cylinder.List.fbAllocateRobot_LeftClamp1(xDone =>,
                                         xBusy =>,
                                         xError =>CylinderStatus.AllocateRobot_LeftClamp1.Error,
                                         xEnable :=,
                                         FrontSensor :=,
                                         RearSensor :=,
                                         SetupPara := CurrentData.Cylinders.AllocateRobot_LeftClamp1,
                                         CurrentCylinderType =>,
                                         InFrontPosition =>CylinderStatus.AllocateRobot_LeftClamp1.InFrontPosition,
                                         InRearPosition =>CylinderStatus.AllocateRobot_LeftClamp1.InRearPosition,
                                         ExtendOutput => InternalOutput.bAllocateRobot_LeftClamp1_Close_Valve,
                                         RetractOutput => InternalOutput.bAllocateRobot_LeftClamp1_Open_Valve);
cylinder.List.fbAllocateRobot_LeftClamp1.IsDoubleValve := TRUE;

cylinder.List.fbAllocateRobot_LeftClamp2(xDone =>,
                                         xBusy =>,
                                         xError =>CylinderStatus.AllocateRobot_LeftClamp2.Error,
                                         xEnable :=,
                                         FrontSensor :=,
                                         RearSensor :=,
                                         SetupPara := CurrentData.Cylinders.AllocateRobot_LeftClamp2,
                                         CurrentCylinderType =>,
                                         InFrontPosition =>CylinderStatus.AllocateRobot_LeftClamp2.InFrontPosition,
                                         InRearPosition =>CylinderStatus.AllocateRobot_LeftClamp2.InRearPosition,
                                         ExtendOutput => InternalOutput.bAllocateRobot_LeftClamp2_Close_Valve,
                                         RetractOutput => InternalOutput.bAllocateRobot_LeftClamp2_Open_Valve);
cylinder.List.fbAllocateRobot_LeftClamp2.IsDoubleValve := TRUE;

cylinder.List.fbAllocateRobot_RightClamp1(xDone =>,
                                          xBusy =>,
                                          xError =>CylinderStatus.AllocateRobot_RightClamp1.Error,
                                          xEnable :=,
                                          FrontSensor :=,
                                          RearSensor :=,
                                          SetupPara := CurrentData.Cylinders.AllocateRobot_RightClamp1,
                                          CurrentCylinderType =>,
                                          InFrontPosition =>CylinderStatus.AllocateRobot_RightClamp1.InFrontPosition,
                                          InRearPosition =>CylinderStatus.AllocateRobot_RightClamp1.InRearPosition,
                                          ExtendOutput => InternalOutput.bAllocateRobot_RightClamp1_Close_Valve,
                                          RetractOutput => InternalOutput.bAllocateRobot_RightClamp1_Open_Valve);
cylinder.List.fbAllocateRobot_RightClamp1.IsDoubleValve := TRUE;

cylinder.List.fbAllocateRobot_RightClamp2(xDone =>,
                                          xBusy =>,
                                          xError =>CylinderStatus.AllocateRobot_RightClamp2.Error,
                                          xEnable :=,
                                          FrontSensor :=,
                                          RearSensor :=,
                                          SetupPara := CurrentData.Cylinders.AllocateRobot_RightClamp2,
                                          CurrentCylinderType =>,
                                          InFrontPosition =>CylinderStatus.AllocateRobot_RightClamp2.InFrontPosition,
                                          InRearPosition =>CylinderStatus.AllocateRobot_RightClamp2.InRearPosition,
                                          ExtendOutput => InternalOutput.bAllocateRobot_RightClamp2_Close_Valve,
                                          RetractOutput => InternalOutput.bAllocateRobot_RightClamp2_Open_Valve);
cylinder.List.fbAllocateRobot_RightClamp2.IsDoubleValve := TRUE;

cylinder.List.fbRoundBelt_WorkZone_Press(xDone =>,
                                         xBusy =>,
                                         xError =>CylinderStatus.RoundBelt_WorkZone_Press.Error,
                                         xEnable :=,
                                         FrontSensor :=,
                                         RearSensor := input.bRoundBelt_WorkZonePress_RearSensor,
                                         SetupPara := CurrentData.Cylinders.RoundBelt_WorkZone_Press,
                                         CurrentCylinderType =>,
                                         InFrontPosition =>CylinderStatus.RoundBelt_WorkZone_Press.InFrontPosition,
                                         InRearPosition =>CylinderStatus.RoundBelt_WorkZone_Press.InRearPosition,
                                         ExtendOutput => InternalOutput.bRoundBelt_WorkZone_Press_Valve,
                                         RetractOutput =>);

cylinder.List.fbRoundBelt_WorkZone_Plug(xDone =>,
                                        xBusy =>,
                                        xError =>CylinderStatus.RoundBelt_WorkZone_Plug.Error,
                                        xEnable :=,
                                        FrontSensor := input.bRoundBelt_WorkZonePlug_frontSensor,
                                        RearSensor := INPUT.bRoundBelt_WorkZonePlug_RearSensor,
                                        SetupPara := CurrentData.Cylinders.RoundBelt_WorkZone_Plug,
                                        CurrentCylinderType =>,
                                        InFrontPosition =>CylinderStatus.RoundBelt_WorkZone_Plug.InFrontPosition,
                                        InRearPosition =>CylinderStatus.RoundBelt_WorkZone_Plug.InRearPosition,
                                        ExtendOutput => InternalOutput.bRoundBelt_WorkZone_Plug_Valve,
                                        RetractOutput =>);

cylinder.List.fbRoundBelt_ChargeZone_Plug(xDone =>,
                                          xBusy =>,
                                          xError =>CylinderStatus.RoundBelt_ChargeZone_Plug.Error,
                                          xEnable :=,
                                          FrontSensor := INPUT.bRoundBelt_ChangeZonePlug_FrontSensor,
                                          RearSensor := input.bRoundBelt_ChangeZonePlug_RearSensor,
                                          SetupPara := CurrentData.Cylinders.RoundBelt_ChargeZone_Plug,
                                          CurrentCylinderType =>,
                                          InFrontPosition =>CylinderStatus.RoundBelt_ChargeZone_Plug.InFrontPosition,
                                          InRearPosition =>CylinderStatus.RoundBelt_ChargeZone_Plug.InRearPosition,
                                          ExtendOutput => InternalOutput.bRoundBelt_ChargeZone_Plug_Valve,
                                          RetractOutput =>);

cylinder.List.fbRoundBelt_TransmitCVZone_Plug(xDone =>,
                                              xBusy =>,
                                              xError =>CylinderStatus.RoundBelt_TransmitCVZone_Plug.Error,
                                              xEnable :=,
                                              FrontSensor := input.bRoundBelt_TransmitCVZonePlug_FrontSensor,
                                              RearSensor := INPUT.bRoundBelt_TransmitCVZonePlug_RearSensor,
                                              SetupPara := CurrentData.Cylinders.RoundBelt_TransmitCVZone_Plug,
                                              CurrentCylinderType =>,
                                              InFrontPosition =>CylinderStatus.RoundBelt_TransmitCVZone_Plug.InFrontPosition,
                                              InRearPosition =>CylinderStatus.RoundBelt_TransmitCVZone_Plug.InRearPosition,
                                              ExtendOutput => InternalOutput.bRoundBelt_TransmitCVZone_Plug_Valve,
                                              RetractOutput =>);

cylinder.List.fbOutRobot_AsideVert(xDone =>,
                                   xBusy =>,
                                   xError =>CylinderStatus.OutRobot_AsideVert.Error,
                                   xEnable :=,
                                   FrontSensor := INPUT.bOutRobot_AsideVert_LowSensor,
                                   RearSensor := input.bOutRobot_AsideVert_highSensor,
                                   SetupPara := CurrentData.Cylinders.OutRobot_AsideVert,
                                   CurrentCylinderType =>,
                                   InFrontPosition =>CylinderStatus.OutRobot_AsideVert.InFrontPosition,
                                   InRearPosition =>CylinderStatus.OutRobot_AsideVert.InRearPosition,
                                   ExtendOutput => InternalOutput.bOutRobot_AsideVert_Valve,
                                   RetractOutput =>);

cylinder.List.fbOutRobot_BsideVert(xDone =>,
                                   xBusy =>,
                                   xError =>CylinderStatus.OutRobot_BsideVert.Error,
                                   xEnable :=,
                                   FrontSensor := input.bOutRobot_BsideVert_LowSensor,
                                   RearSensor := INPUT.bOutRobot_BsideVert_HighSensor,
                                   SetupPara := CurrentData.Cylinders.OutRobot_BsideVert,
                                   CurrentCylinderType =>,
                                   InFrontPosition =>CylinderStatus.OutRobot_BsideVert.InFrontPosition,
                                   InRearPosition =>CylinderStatus.OutRobot_BsideVert.InRearPosition,
                                   ExtendOutput => InternalOutput.bOutRobot_BsideVert_Valve,
                                   RetractOutput =>);

cylinder.List.fbOutRobot_AsideClamp(xDone =>,
                                    xBusy =>,
                                    xError =>CylinderStatus.OutRobot_AsideClamp.Error,
                                    xEnable :=,
                                    FrontSensor :=,
                                    RearSensor := input.bOutRobot_AsideClamp_RearSensor,
                                    SetupPara := CurrentData.Cylinders.OutRobot_AsideClamp,
                                    CurrentCylinderType =>,
                                    InFrontPosition =>CylinderStatus.OutRobot_AsideClamp.InFrontPosition,
                                    InRearPosition =>CylinderStatus.OutRobot_AsideClamp.InRearPosition,
                                    ExtendOutput => InternalOutput.bOutRobot_AsideClamp_Close_Valve,
                                    RetractOutput => InternalOutput.bOutRobot_AsideClamp_Open_Valve);
cylinder.List.fbOutRobot_AsideClamp.IsDoubleValve := TRUE;

cylinder.List.fbOutRobot_BsideClamp(xDone =>,
                                    xBusy =>,
                                    xError =>CylinderStatus.OutRobot_BsideClamp.Error,
                                    xEnable :=,
                                    FrontSensor :=,
                                    RearSensor := input.bOutRobot_BsideClamp_RearSensor,
                                    SetupPara := CurrentData.Cylinders.OutRobot_BsideClamp,
                                    CurrentCylinderType =>,
                                    InFrontPosition =>CylinderStatus.OutRobot_BsideClamp.InFrontPosition,
                                    InRearPosition =>CylinderStatus.OutRobot_BsideClamp.InRearPosition,
                                    ExtendOutput => InternalOutput.bOutRobot_BsideClamp_Close_Valve,
                                    RetractOutput => InternalOutput.bOutRobot_BsideClamp_Open_Valve);
cylinder.List.fbOutRobot_BsideClamp.IsDoubleValve := TRUE;

cylinder.List.fbTransmitCV_CamaraHoriz(xDone =>,
                                       xBusy =>,
                                       xError =>CylinderStatus.TransmitCV_CamaraHoriz.Error,
                                       xEnable :=,
                                       FrontSensor :=input.bTransmit_CamaraHorizDifferentSizeSide_Sensor,
                                       RearSensor := input.bTransmit_CamaraHorizSameSizeSide_Sensor,
                                       SetupPara := CurrentData.Cylinders.TransmitCV_CamaraHoriz,
                                       CurrentCylinderType =>,
                                       InFrontPosition =>CylinderStatus.TransmitCV_CamaraHoriz.InFrontPosition,
                                       InRearPosition =>CylinderStatus.TransmitCV_CamaraHoriz.InRearPosition,
                                       ExtendOutput => InternalOutput.bTransmitCV_CamaraHorizDifferentSide_Valve,
                                       RetractOutput => InternalOutput.bTransmitCV_CamaraHorizSameSizeSide_Valve);
cylinder.List.fbTransmitCV_CamaraHoriz.IsDoubleValve := TRUE;

cylinder.List.fbDifferentSizeCV_Press2(xDone =>,
                                       xBusy =>,
                                       xError =>CylinderStatus.DifferentSizeCV_Press2.Error,
                                       xEnable :=,
                                       FrontSensor :=,
                                       RearSensor :=,
                                       SetupPara := CurrentData.Cylinders.DifferentSizeCV_Press2,
                                       CurrentCylinderType =>,
                                       InFrontPosition =>CylinderStatus.DifferentSizeCV_Press2.InFrontPosition,
                                       InRearPosition =>CylinderStatus.DifferentSizeCV_Press2.InRearPosition,
                                       ExtendOutput => InternalOutput.bDifferentSizeCV_Press2_Valve,
                                       RetractOutput =>);

cylinder.List.fbDifferentSizeCV_Press1(xDone =>,
                                       xBusy =>,
                                       xError =>CylinderStatus.DifferentSizeCV_Press1.Error,
                                       xEnable :=,
                                       FrontSensor :=,
                                       RearSensor :=,
                                       SetupPara := CurrentData.Cylinders.DifferentSizeCV_Press1,
                                       CurrentCylinderType =>,
                                       InFrontPosition =>CylinderStatus.DifferentSizeCV_Press1.InFrontPosition,
                                       InRearPosition =>CylinderStatus.DifferentSizeCV_Press1.InRearPosition,
                                       ExtendOutput => InternalOutput.bDifferentSizeCV_Press1_Valve,
                                       RetractOutput =>);

cylinder.List.fbDifferentSizeCV_Block1(xDone =>,
                                       xBusy =>,
                                       xError =>CylinderStatus.DifferentSizeCV_Block1.Error,
                                       xEnable :=,
                                       FrontSensor :=,
                                       RearSensor := INPUT.bDifferentCV_Block_RearSensor,
                                       SetupPara := CurrentData.Cylinders.DifferentSizeCV_Block1,
                                       CurrentCylinderType =>,
                                       InFrontPosition =>CylinderStatus.DifferentSizeCV_Block1.InFrontPosition,
                                       InRearPosition =>CylinderStatus.DifferentSizeCV_Block1.InRearPosition,
                                       ExtendOutput => InternalOutput.bDifferentSizeCV_Block1_Valve,
                                       RetractOutput =>);

cylinder.List.fbSameSizeCV_Press4(xDone =>,
                                  xBusy =>,
                                  xError =>CylinderStatus.SameSizeCV_Press4.Error,
                                  xEnable :=,
                                  FrontSensor :=,
                                  RearSensor :=,
                                  SetupPara := CurrentData.Cylinders.SameSizeCV_Press4,
                                  CurrentCylinderType =>,
                                  InFrontPosition =>CylinderStatus.SameSizeCV_Press4.InFrontPosition,
                                  InRearPosition =>CylinderStatus.SameSizeCV_Press4.InRearPosition,
                                  ExtendOutput => InternalOutput.bSameSizeCV_Press4_Valve,
                                  RetractOutput =>);

cylinder.List.fbSameSizeCV_Press3(xDone =>,
                                  xBusy =>,
                                  xError =>CylinderStatus.SameSizeCV_Press3.Error,
                                  xEnable :=,
                                  FrontSensor :=,
                                  RearSensor :=,
                                  SetupPara := CurrentData.Cylinders.SameSizeCV_Press3,
                                  CurrentCylinderType =>,
                                  InFrontPosition =>CylinderStatus.SameSizeCV_Press3.InFrontPosition,
                                  InRearPosition =>CylinderStatus.SameSizeCV_Press3.InRearPosition,
                                  ExtendOutput => InternalOutput.bSameSizeCV_Press3_Valve,
                                  RetractOutput =>);

cylinder.List.fbSameSizeCV_Press2(xDone =>,
                                  xBusy =>,
                                  xError =>CylinderStatus.SameSizeCV_Press2.Error,
                                  xEnable :=,
                                  FrontSensor :=,
                                  RearSensor :=,
                                  SetupPara := CurrentData.Cylinders.SameSizeCV_Press2,
                                  CurrentCylinderType =>,
                                  InFrontPosition =>CylinderStatus.SameSizeCV_Press2.InFrontPosition,
                                  InRearPosition =>CylinderStatus.SameSizeCV_Press2.InRearPosition,
                                  ExtendOutput => InternalOutput.bSameSizeCV_Press2_Valve,
                                  RetractOutput =>);

cylinder.List.fbSameSizeCV_Press1(xDone =>,
                                  xBusy =>,
                                  xError =>CylinderStatus.SameSizeCV_Press1.Error,
                                  xEnable :=,
                                  FrontSensor :=,
                                  RearSensor :=,
                                  SetupPara := CurrentData.Cylinders.SameSizeCV_Press1,
                                  CurrentCylinderType =>,
                                  InFrontPosition =>CylinderStatus.SameSizeCV_Press1.InFrontPosition,
                                  InRearPosition =>CylinderStatus.SameSizeCV_Press1.InRearPosition,
                                  ExtendOutput => InternalOutput.bSameSizeCV_Press1_Valve,
                                  RetractOutput =>);

cylinder.List.fbSameSizeCV_Block2(xDone =>,
                                  xBusy =>,
                                  xError =>CylinderStatus.SameSizeCV_Block2.Error,
                                  xEnable :=,
                                  FrontSensor :=,
                                  RearSensor := input.bSameSizeCVBlock2_RearSensor,
                                  SetupPara := CurrentData.Cylinders.SameSizeCV_Block2,
                                  CurrentCylinderType =>,
                                  InFrontPosition =>CylinderStatus.SameSizeCV_Block2.InFrontPosition,
                                  InRearPosition =>CylinderStatus.SameSizeCV_Block2.InRearPosition,
                                  ExtendOutput => InternalOutput.bSameSizeCV_Block2_Valve,
                                  RetractOutput =>);

cylinder.List.fbSameSizeCV_Block1(xDone =>,
                                  xBusy =>,
                                  xError =>CylinderStatus.SameSizeCV_Block1.Error,
                                  xEnable :=,
                                  FrontSensor :=,
                                  RearSensor := input.bSameSizeCVBlock1_RearSensor,
                                  SetupPara := CurrentData.Cylinders.SameSizeCV_Block1,
                                  CurrentCylinderType =>,
                                  InFrontPosition =>CylinderStatus.SameSizeCV_Block1.InFrontPosition,
                                  InRearPosition =>CylinderStatus.SameSizeCV_Block1.InRearPosition,
                                  ExtendOutput => InternalOutput.bSameSizeCV_Block1_Valve,
                                  RetractOutput =>);

cylinder.List.fbTurntable_Press(xDone =>,
                                xBusy =>,
                                xError =>CylinderStatus.Turntable_Press.Error,
                                xEnable :=,
                                FrontSensor :=,
                                RearSensor := input.bTurnTable_Press_RearSensor,
                                SetupPara := CurrentData.Cylinders.Turntable_Press,
                                CurrentCylinderType =>,
                                InFrontPosition =>CylinderStatus.Turntable_Press.InFrontPosition,
                                InRearPosition =>CylinderStatus.Turntable_Press.InRearPosition,
                                ExtendOutput => InternalOutput.bTurntable_Press_Valve,
                                RetractOutput =>);
Cylinder.List.fbShippingBuffer_Press(xDone=> , 
										xBusy=> , 
										xError=> , 
										xEnable:= , 
										FrontSensor:= , 
										RearSensor:= TRUE, 
										SetupPara:= , 
										CurrentCylinderType=> , 
										InFrontPosition=> , 
										InRearPosition=> , 
										ExtendOutput=> , 
										RetractOutput=> , 
										iErrorID=> , 
										ErrorMsg=> );
END_ACTION

ACTION A02_Motor:
Motor.List.WareHouseCV_10(xDone =>,
                          xBusy =>,
                          xError => MotorStatus.WareHouseCV_10.Error,
                          xEnable :=,
                          OverLoadSignal :=,
                          SetupPara :=,
                          InForWard =>MotorStatus.WareHouseCV_10.InForward,
                          InBackWard =>MotorStatus.WareHouseCV_10.InBackward,
                          InStopped =>MotorStatus.WareHouseCV_10.InStopped,
                          ForWardOutput => InternalOutput.bWareHouseCV10_Fwd,
                          BackWardOutput => InternalOutput.bWareHouseCV10_Rev);

Motor.List.WareHouseCV_09(xDone =>,
                          xBusy =>,
                          xError =>MotorStatus.WareHouseCV_09.Error,
                          xEnable :=,
                          OverLoadSignal :=,
                          SetupPara :=,
                          InForWard =>MotorStatus.WareHouseCV_09.InForward,
                          InBackWard =>MotorStatus.WareHouseCV_09.InBackward,
                          InStopped =>MotorStatus.WareHouseCV_09.InStopped,
                          ForWardOutput =>InternalOutput.bWareHouseCV9_Fwd,
                          BackWardOutput =>InternalOutput.bWareHouseCV9_Rev);

Motor.List.WareHouseCV_08(xDone =>,
                          xBusy =>,
                          xError =>MotorStatus.WareHouseCV_08.Error,
                          xEnable :=,
                          OverLoadSignal :=,
                          SetupPara :=,
                          InForWard =>MotorStatus.WareHouseCV_08.InForward,
                          InBackWard =>MotorStatus.WareHouseCV_08.InBackward,
                          InStopped =>MotorStatus.WareHouseCV_08.InStopped,
                          ForWardOutput =>InternalOutput.bWareHouseCV8_Fwd,
                          BackWardOutput =>InternalOutput.bWareHouseCV8_Rev);

Motor.List.WareHouseCV_07(xDone =>,
                          xBusy =>,
                          xError =>MotorStatus.WareHouseCV_07.Error,
                          xEnable :=,
                          OverLoadSignal :=,
                          SetupPara :=,
                          InForWard =>MotorStatus.WareHouseCV_07.InForward,
                          InBackWard =>MotorStatus.WareHouseCV_07.InBackward,
                          InStopped =>MotorStatus.WareHouseCV_07.InStopped,
                          ForWardOutput =>InternalOutput.bWareHouseCV7_Fwd,
                          BackWardOutput =>InternalOutput.bWareHouseCV7_Rev);

Motor.List.WareHouseCV_06(xDone =>,
                          xBusy =>,
                          xError =>MotorStatus.WareHouseCV_06.Error,
                          xEnable :=,
                          OverLoadSignal :=,
                          SetupPara :=,
                          InForWard =>MotorStatus.WareHouseCV_06.InForward,
                          InBackWard =>MotorStatus.WareHouseCV_06.InBackward,
                          InStopped =>MotorStatus.WareHouseCV_06.InStopped,
                          ForWardOutput =>InternalOutput.bWareHouseCV6_Fwd,
                          BackWardOutput =>InternalOutput.bWareHouseCV6_Rev);

Motor.List.WareHouseCV_05(xDone =>,
                          xBusy =>,
                          xError =>MotorStatus.WareHouseCV_05.Error,
                          xEnable :=,
                          OverLoadSignal :=,
                          SetupPara :=,
                          InForWard =>MotorStatus.WareHouseCV_05.InForward,
                          InBackWard =>MotorStatus.WareHouseCV_05.InBackward,
                          InStopped =>MotorStatus.WareHouseCV_05.InStopped,
                          ForWardOutput =>InternalOutput.bWareHouseCV5_Fwd,
                          BackWardOutput =>InternalOutput.bWareHouseCV5_Rev);

Motor.List.WareHouseCV_04(xDone =>,
                          xBusy =>,
                          xError =>MotorStatus.WareHouseCV_04.Error,
                          xEnable :=,
                          OverLoadSignal :=,
                          SetupPara :=,
                          InForWard =>MotorStatus.WareHouseCV_04.InForward,
                          InBackWard =>MotorStatus.WareHouseCV_04.InBackward,
                          InStopped =>MotorStatus.WareHouseCV_04.InStopped,
                          ForWardOutput =>InternalOutput.bWareHouseCV4_Fwd,
                          BackWardOutput =>InternalOutput.bWareHouseCV4_Rev);

Motor.List.WareHouseCV_03(xDone =>,
                          xBusy =>,
                          xError =>MotorStatus.WareHouseCV_03.Error,
                          xEnable :=,
                          OverLoadSignal :=,
                          SetupPara :=,
                          InForWard =>MotorStatus.WareHouseCV_03.InForward,
                          InBackWard =>MotorStatus.WareHouseCV_03.InBackward,
                          InStopped =>MotorStatus.WareHouseCV_03.InStopped,
                          ForWardOutput =>InternalOutput.bWareHouseCV3_Fwd,
                          BackWardOutput =>InternalOutput.bWareHouseCV3_Rev);

Motor.List.WareHouseCV_02(xDone =>,
                          xBusy =>,
                          xError =>MotorStatus.WareHouseCV_02.Error,
                          xEnable :=,
                          OverLoadSignal :=,
                          SetupPara :=,
                          InForWard =>MotorStatus.WareHouseCV_02.InForward,
                          InBackWard =>MotorStatus.WareHouseCV_02.InBackward,
                          InStopped =>MotorStatus.WareHouseCV_02.InStopped,
                          ForWardOutput =>InternalOutput.bWareHouseCV2_Fwd,
                          BackWardOutput =>InternalOutput.bWareHouseCV2_Rev);

Motor.List.WareHouseCV_01(xDone =>,
                          xBusy =>,
                          xError =>MotorStatus.WareHouseCV_01.Error,
                          xEnable :=,
                          OverLoadSignal :=,
                          SetupPara :=,
                          InForWard =>MotorStatus.WareHouseCV_01.InForward,
                          InBackWard =>MotorStatus.WareHouseCV_01.InBackward,
                          InStopped =>MotorStatus.WareHouseCV_01.InStopped,
                          ForWardOutput =>InternalOutput.bWareHouseCV1_Fwd,
                          BackWardOutput =>InternalOutput.bWareHouseCV1_Rev);

Motor.List.WareHouseCV_20(xDone =>,
                          xBusy =>,
                          xError =>MotorStatus.WareHouseCV_20.Error,
                          xEnable :=,
                          OverLoadSignal :=,
                          SetupPara :=,
                          InForWard =>MotorStatus.WareHouseCV_20.InForward,
                          InBackWard =>MotorStatus.WareHouseCV_20.InBackward,
                          InStopped =>MotorStatus.WareHouseCV_20.InStopped,
                          ForWardOutput =>InternalOutput.bWareHouseCV20_Fwd,
                          BackWardOutput =>InternalOutput.bWareHouseCV20_Rev);

Motor.List.WareHouseCV_19(xDone =>,
                          xBusy =>,
                          xError =>MotorStatus.WareHouseCV_19.Error,
                          xEnable :=,
                          OverLoadSignal :=,
                          SetupPara :=,
                          InForWard =>MotorStatus.WareHouseCV_19.InForward,
                          InBackWard =>MotorStatus.WareHouseCV_19.InBackward,
                          InStopped =>MotorStatus.WareHouseCV_19.InStopped,
                          ForWardOutput =>InternalOutput.bWareHouseCV19_Fwd,
                          BackWardOutput =>InternalOutput.bWareHouseCV19_Rev);

Motor.List.WareHouseCV_18(xDone =>,
                          xBusy =>,
                          xError =>MotorStatus.WareHouseCV_18.Error,
                          xEnable :=,
                          OverLoadSignal :=,
                          SetupPara :=,
                          InForWard =>MotorStatus.WareHouseCV_18.InForward,
                          InBackWard =>MotorStatus.WareHouseCV_18.InBackward,
                          InStopped =>MotorStatus.WareHouseCV_18.InStopped,
                          ForWardOutput =>InternalOutput.bWareHouseCV18_Fwd,
                          BackWardOutput =>InternalOutput.bWareHouseCV18_Rev);

Motor.List.WareHouseCV_17(xDone =>,
                          xBusy =>,
                          xError =>MotorStatus.WareHouseCV_17.Error,
                          xEnable :=,
                          OverLoadSignal :=,
                          SetupPara :=,
                          InForWard =>MotorStatus.WareHouseCV_17.InForward,
                          InBackWard =>MotorStatus.WareHouseCV_17.InBackward,
                          InStopped =>MotorStatus.WareHouseCV_17.InStopped,
                          ForWardOutput =>InternalOutput.bWareHouseCV17_Fwd,
                          BackWardOutput =>InternalOutput.bWareHouseCV17_Rev);

Motor.List.WareHouseCV_16(xDone =>,
                          xBusy =>,
                          xError =>MotorStatus.WareHouseCV_16.Error,
                          xEnable :=,
                          OverLoadSignal :=,
                          SetupPara :=,
                          InForWard =>MotorStatus.WareHouseCV_16.InForward,
                          InBackWard =>MotorStatus.WareHouseCV_16.InBackward,
                          InStopped =>MotorStatus.WareHouseCV_16.InStopped,
                          ForWardOutput =>InternalOutput.bWareHouseCV16_Fwd,
                          BackWardOutput =>InternalOutput.bWareHouseCV16_Rev);

Motor.List.WareHouseCV_15(xDone =>,
                          xBusy =>,
                          xError =>MotorStatus.WareHouseCV_15.Error,
                          xEnable :=,
                          OverLoadSignal :=,
                          SetupPara :=,
                          InForWard =>MotorStatus.WareHouseCV_15.InForward,
                          InBackWard =>MotorStatus.WareHouseCV_15.InBackward,
                          InStopped =>MotorStatus.WareHouseCV_15.InStopped,
                          ForWardOutput =>InternalOutput.bWareHouseCV15_Fwd,
                          BackWardOutput =>InternalOutput.bWareHouseCV15_Rev);

Motor.List.WareHouseCV_14(xDone =>,
                          xBusy =>,
                          xError =>MotorStatus.WareHouseCV_14.Error,
                          xEnable :=,
                          OverLoadSignal :=,
                          SetupPara :=,
                          InForWard =>MotorStatus.WareHouseCV_14.InForward,
                          InBackWard =>MotorStatus.WareHouseCV_14.InBackward,
                          InStopped =>MotorStatus.WareHouseCV_14.InStopped,
                          ForWardOutput =>InternalOutput.bWareHouseCV14_Fwd,
                          BackWardOutput =>InternalOutput.bWareHouseCV14_Rev);

Motor.List.WareHouseCV_13(xDone =>,
                          xBusy =>,
                          xError =>MotorStatus.WareHouseCV_13.Error,
                          xEnable :=,
                          OverLoadSignal :=,
                          SetupPara :=,
                          InForWard =>MotorStatus.WareHouseCV_13.InForward,
                          InBackWard =>MotorStatus.WareHouseCV_13.InBackward,
                          InStopped =>MotorStatus.WareHouseCV_13.InStopped,
                          ForWardOutput =>InternalOutput.bWareHouseCV13_Fwd,
                          BackWardOutput =>InternalOutput.bWareHouseCV13_Rev);

Motor.List.WareHouseCV_12(xDone =>,
                          xBusy =>,
                          xError =>MotorStatus.WareHouseCV_12.Error,
                          xEnable :=,
                          OverLoadSignal :=,
                          SetupPara :=,
                          InForWard =>MotorStatus.WareHouseCV_12.InForward,
                          InBackWard =>MotorStatus.WareHouseCV_12.InBackward,
                          InStopped =>MotorStatus.WareHouseCV_12.InStopped,
                          ForWardOutput =>InternalOutput.bWareHouseCV12_Fwd,
                          BackWardOutput =>InternalOutput.bWareHouseCV12_Rev);

Motor.List.WareHouseCV_11(xDone =>,
                          xBusy =>,
                          xError =>MotorStatus.WareHouseCV_11.Error,
                          xEnable :=,
                          OverLoadSignal :=,
                          SetupPara :=,
                          InForWard =>MotorStatus.WareHouseCV_11.InForward,
                          InBackWard =>MotorStatus.WareHouseCV_11.InBackward,
                          InStopped =>MotorStatus.WareHouseCV_11.InStopped,
                          ForWardOutput =>InternalOutput.bWareHouseCV11_Fwd,
                          BackWardOutput =>InternalOutput.bWareHouseCV11_Rev);

Motor.List.UpCV(xDone =>,
                xBusy =>,
                xError =>MotorStatus.UpCV.Error,
                xEnable :=,
                OverLoadSignal :=,
                SetupPara :=,
                InForWard =>MotorStatus.UpCV.InForward,
                InBackWard =>MotorStatus.UpCV.InBackward,
                InStopped =>MotorStatus.UpCV.InStopped,
                ForWardOutput =>InternalOutput.bUpCV_Fwd,
                BackWardOutput =>InternalOutput.bUpCV_Rev);

Motor.List.LowCV(xDone =>,
                xBusy =>,
                xError =>MotorStatus.LowCV.Error,
                xEnable :=,
                OverLoadSignal :=,
                SetupPara :=,
                InForWard =>MotorStatus.LowCV.InForward,
                InBackWard =>MotorStatus.LowCV.InBackward,
                InStopped =>MotorStatus.LowCV.InStopped,
                ForWardOutput =>InternalOutput.bLowCV_Fwd,
                BackWardOutput =>InternalOutput.bLowCV_Rev);

Motor.List.PullOutCV_A(xDone =>,
						xBusy =>,
						xError =>MotorStatus.PullOutCV_A.Error,
						xEnable :=,
						OverLoadSignal :=,
						SetupPara :=,
						InForWard =>MotorStatus.PullOutCV_A.InForward,
						InBackWard =>MotorStatus.PullOutCV_A.InBackward,
						InStopped =>MotorStatus.PullOutCV_A.InStopped,
						ForWardOutput =>InternalOutput.bPullOutCV_A_Fwd,
						BackWardOutput =>InternalOutput.bPullOutCV_A_Rev);

Motor.List.PullOutCV_B(xDone =>,
						xBusy =>,
						xError =>MotorStatus.PullOutCV_B.Error,
						xEnable :=,
						OverLoadSignal :=,
						SetupPara :=,
						InForWard =>MotorStatus.PullOutCV_B.InForward,
						InBackWard =>MotorStatus.PullOutCV_B.InBackward,
						InStopped =>MotorStatus.PullOutCV_B.InStopped,
						ForWardOutput =>InternalOutput.bPullOutCV_B_Fwd,
						BackWardOutput =>InternalOutput.bPullOutCV_B_Rev);

Motor.List.TransmitSameSideCV(xDone =>,
								xBusy =>,
								xError =>MotorStatus.TransmitSameSideCV.Error,
								xEnable :=,
								OverLoadSignal :=,
								SetupPara :=,
								InForWard =>MotorStatus.TransmitSameSideCV.InForward,
								InBackWard =>MotorStatus.TransmitSameSideCV.InBackward,
								InStopped =>MotorStatus.TransmitSameSideCV.InStopped,
								ForWardOutput =>InternalOutput.bTransmitCV_SameSizeSide_Fwd,
								BackWardOutput =>InternalOutput.bTransmitCV_SameSide_Rev);

Motor.List.TransmitDifferentSideCV(xDone =>,
									xBusy =>,
									xError =>MotorStatus.TransmitDifferentSideCV.Error,
									xEnable :=,
									OverLoadSignal :=,
									SetupPara :=,
									InForWard =>MotorStatus.TransmitDifferentSideCV.InForward,
									InBackWard =>MotorStatus.TransmitDifferentSideCV.InBackward,
									InStopped =>MotorStatus.TransmitDifferentSideCV.InStopped,
									ForWardOutput =>InternalOutput.bTransmitCV_DifferentSide_Fwd,
									BackWardOutput =>InternalOutput.bTransmitCV_DifferentSide_Rev);
END_ACTION

ACTION A03_FanucRobot:
FanucRobot.List.StorageRobot(
	Estop:= Machine_Estop (*OR Input.bStorage_EstopPb*), 
	OpMode:= , 
	Start:= Machine_Start OR RobotService_StartCmd , 
//	Reset:= Machine_Reset OR fbStorageArea.RobotResetCMD, 
//	Hold:= Machine_Stop, 
	Reset:= Machine_Reset OR fbStorageArea.RobotResetCMD OR tofResetDelay.Q OR RobotService_ResetCmd, //Postpone reset signal to fanuc robot		
	Hold:=   NOT FanucRobot.List.StorageRobot.Error AND_THEN Machine_Stop, 		//Transport form Kinsus version to taixin
	ManualCtrl :=  GVL_HMI.Storage.Manual.FanucRobot,
            SimMode    := EnableSimulation,
        	qEnable=> , 
        	qFault=> ,

        	E_Stop_Output=> StorageRobot_EStop, 
        	Halt=> , 
        	Error=> , 
        	ErrorID=> );

        FanucRobot.List.ShippingRobot(
        	Estop:= Machine_Estop (*OR Input.bStorage_EstopPb*), 
        	OpMode:= , 
        	Start:= Machine_Start OR ShippingRobotService_StartCmd, 
        	Reset:= Machine_Reset OR fbShippingArea.RobotResetCMD OR tofResetDelay.Q OR ShippingRobotService_ResetCmd, 			//
        	Hold:= NOT fanucrobot.List.ShippingRobot.Error AND_THEN Machine_Stop,
        	ManualCtrl:= GVL_HMI.Shipping.Manual.FanucRobot,
            SimMode    := EnableSimulation,
        	qEnable=> , 
        	qFault=> , 
        	E_Stop_Output=> ShippingRobot_EStop, 
        	Halt=> , 
        	Error=> , 
        	ErrorID=> );
END_ACTION

ACTION A04_OpPannel:
// E-Stop 
Machine_Estop := (NOT INPUT.bAllocate_EStopPb OR
                 NOT INPUT.bStorage_EstopPb OR
                 StorageRobot_EStop OR
                 ShippingRobot_EStop OR
                 GVL_ADS.OpPannel_Ctrl.EStopBtnStatus OR 
				NOT INPUT.bStorage_AirPressure_Ready) AND
                 NOT EnableSimulation;

// Stop
bSafetyDoorOpen := (NOT INPUT.bSafetyDoor1 OR
                   NOT INPUT.bSafetyDoor2 OR
                   NOT INPUT.bSafetyDoor3 OR
                   NOT INPUT.bSafetyDoor4 OR		
                   NOT INPUT.bSafetyDoor5 OR
                   NOT INPUT.bSafetyDoor6 OR
                   NOT INPUT.bSafetyDoor7 OR
                   NOT INPUT.bSafetyDoor8 OR
                   not INPUT.bSafetyDoor9 OR
                   not INPUT.bSafetyDoor10 OR
                   not INPUT.bSafetyDoor11 OR
                   not INPUT.bSafetyDoor12 OR
                   not INPUT.bSafetyDoor13 OR
                   not INPUT.bSafetyDoor14 OR
                   NOT INPUT.bAllocate_Electrical_Cabinet_SafetyDoor OR
                   NOT INPUT.bShippingRobot_ElectricalCabinet_SafetyDoor) AND
				   (NOT    GVL_HMI.Setup.Mechanical.stSafetyByPass.SafeDoorByPass)	;		//use Safedoor bypass

// 暫停復位 需要按下reset 之後start 後續做。	//edited by Gamin 20260202
IF StopEdgeDetect.xRisingEdge THEN
    bStopMem 	:= TRUE;
	ResetDetect := FALSE;
ELSIF ResetEdgeDetect.xRisingEdge THEN
//  bStopMem 	:= FALSE;
	ResetDetect := TRUE;
ELSIF StartEdgeDetect.xRisingEdge AND ResetDetect THEN
	bStopMem 	:= FALSE;
END_IF

Machine_Stop := (INPUT.bAllocate_StopPb OR
                INPUT.bStorage_StopPb OR
                bSafetyDoorOpen OR
                xError OR
                GVL_ADS.OpPannel_Ctrl.StopBtnStatus)
				AND NOT (eStateCurrent = ePMLState_Aborted);;

// Reset
Machine_Reset :=
    INPUT.bAllocate_ResetPb OR INPUT.bStorage_ResetPb OR GVL_ADS.OpPannel_Ctrl.ResetBtnStatus;

// Start
Machine_Start :=
    INPUT.bAllocate_StartPb OR INPUT.bStorage_StartPb OR GVL_ADS.OpPannel_Ctrl.StartBtnStatus;

//IF xError THEN
//    InternalOutput.bAllocated_SignalTower_RedLamp := fbBlink_05.OUT;
//    InternalOutput.bStorage_SingleTower_RedLamp := fbBlink_05.OUT;
//	InternalOutput.bAllocated_StopPbLamp := fbBlink_05.OUT;
//	InternalOutput.bStorage_StopPbLamp := fbBlink_05.OUT;
//ELSIF bStopMem AND NOT xError THEN
//    InternalOutput.bAllocated_SignalTower_RedLamp := TRUE;
//    InternalOutput.bStorage_SingleTower_RedLamp := TRUE;
//	InternalOutput.bAllocated_StopPbLamp := TRUE;
//	InternalOutput.bStorage_StopPbLamp := TRUE;
//ELSE
//    InternalOutput.bAllocated_SignalTower_RedLamp := FALSE;
//    InternalOutput.bStorage_SingleTower_RedLamp := FALSE;
//	InternalOutput.bAllocated_StopPbLamp := FALSE;
//	InternalOutput.bStorage_StopPbLamp := FALSE;

//END_IF

InternalOutput.bAllocated_SignalTower_RedLamp := _RedLamp;
InternalOutput.bAllocated_SignalTower_YellowLamp := _YellowLamp;
InternalOutput.bAllocated_SignalTower_GreenLamp := _GreenLamp;
InternalOutput.bAllocated_Buzzer := _Buzz OR BuzzCtrlUseBuzz;
InternalOutput.bStorage_Buzzer 	 := _Buzz OR BuzzCtrlUseBuzz;
InternalOutput.bStorage_SingleTower_RedLamp := _RedLamp;
InternalOutput.bStorage_SingleTower_YellowLamp := _YellowLamp;
InternalOutput.bStorage_SingleTower_GreenLamp := _GreenLamp;

InternalOutput.bAllocated_StopPbLamp := _RedLamp;
InternalOutput.bAllocated_StartPbLamp := _GreenLamp;
InternalOutput.bAllocated_ResetPbLamp := _YellowLamp;

InternalOutput.bStorage_ResetPbLamp := _YellowLamp;
InternalOutput.bStorage_StartPbLamp := _GreenLamp;
InternalOutput.bStorage_StopPbLamp := _RedLamp;

//postpone btn signal to Host
tofResetDelay.IN:=Machine_Reset;
tofStopDelay.IN :=Machine_Stop; 
tofStartDelay.IN:=Machine_Start;
tofResetDelay(PT:=T#3.2S);	
tofStopDelay(PT:=T#1S);	
tofStartDelay(PT:=T#1S);

GVL_ADS.OpPannel_Status.EStopBtnStatus := Machine_Estop;
GVL_ADS.OpPannel_Status.ResetBtnStatus := tofResetDelay.Q;
GVL_ADS.OpPannel_Status.StartBtnStatus := tofStartDelay.Q;
GVL_ADS.OpPannel_Status.StopBtnStatus  := tofStopDelay.Q OR bStopMem;


fb_AllocateSignalTower(
	Enable:= , 
	LampRed:= _RedLamp, 
	LampYellow:= _YellowLamp, 
	LampGreen:= _GreenLamp, 
	Buzz:= _Buzz, 
	ForceCloseBuzz:= , 
	BuzzSwitchOnTime:= 30000, 
	//BuzzSwitchOnTime:= 2, 
	Vaild=> , 
	Error=> , 
	ErrorID=> );
END_ACTION

ACTION A05_Light:
//  Light 
InternalOutput.bStorage_EleBoxLight := GVL_HMI.Setup.Light.Storage_EleBoxLight_Off;
InternalOutput.bStorage_AreaLight := GVL_HMI.Setup.Light.Storage_AreaLight_Off;
InternalOutput.bAllocated_AreaLight := GVL_HMI.Setup.Light.Allocated_AreaLight_Off;

// Upcv CameraBlow
//InternalOutput.bCamara_Blow := GVL_HMI.Storage.Manual.UpCV.CameraBlow;
IF fbHmiCameraBlow.xRisingEdge THEN
	InternalOutput.bCamara_Blow := TRUE;
ELSIF fbHmiCameraBlow.xFallingEdge THEN
	InternalOutput.bCamara_Blow := FALSE;
END_IF
END_ACTION

ACTION A10_ErrorHandler:
IF NOT ErrorTableInitDone THEN
	ErrorTableInitDone := M_General_AlarmRegister();
END_IF
M_General_AlarmRegister();
//Machine_Estop := ( NOT INPUT.bAllocate_EStopPb (*OR INPUT.bStorage_EstopPb*) OR StorageRobot_EStop OR ShippingRobot_EStop)  AND NOT EnableSimulation ;
E_StopEdgeDetect(xInput := Machine_Estop);
ResetEdgeDetect(xInput:= Machine_Reset);
StopEdgeDetect(xInput:= Machine_Stop);
StartEdgeDetect(xInput:= Machine_Start);

IF Allocate_EStopEdgeDetect.xRisingEdge THEN
	Allocate_EStop := FALSE;
ELSIF Allocate_EStopEdgeDetect.xFallingEdge THEN
	Allocate_EStop := TRUE;
END_IF

IF Storage_EstopEdgeDetect.xRisingEdge THEN
	Storage_EStop := FALSE;
ELSIF Storage_EstopEdgeDetect.xFallingEdge THEN
	Storage_EStop := TRUE;
END_IF

IF fbErrorHandler.ActiveAlarmCount <> 0 THEN
    xError := TRUE;
ELSE
    xError := FALSE;
END_IF

CASE fbErrorHandler.CurrentSeverityLevel OF
	E_Severity.Level7,E_Severity.Level6:
		IF xError AND (PackTag.Status.StateCurrent <> ePMLState_Aborted) THEN
			PackTag.Command.CntrlCmd := ePMLCommand_Abort;
		END_IF
END_CASE

IF ResetEdgeDetect.xRisingEdge THEN
//////////// Axis
	IF arAxisCtrl_gb[AxisNo.Allocate_X].Admin.Axis.Status.Error THEN
		arAxisCtrl_gb[AxisNo.Allocate_X].Admin.ClearError := Machine_Reset;
	END_IF
	IF arAxisCtrl_gb[AxisNo.Allocate_Y].Admin.Axis.Status.Error THEN
		arAxisCtrl_gb[AxisNo.Allocate_Y].Admin.ClearError := Machine_Reset;
	END_IF
	IF arAxisCtrl_gb[AxisNo.OutRobot_X].Admin.Axis.Status.Error THEN
		arAxisCtrl_gb[AxisNo.OutRobot_X].Admin.ClearError := Machine_Reset;
	END_IF
	IF arAxisCtrl_gb[AxisNo.OutRobot_Y].Admin.Axis.Status.Error THEN
		arAxisCtrl_gb[AxisNo.OutRobot_Y].Admin.ClearError := Machine_Reset;
	END_IF
	IF arAxisCtrl_gb[AxisNo.RoundBelt].Admin.Axis.Status.Error THEN
		arAxisCtrl_gb[AxisNo.RoundBelt].Admin.ClearError := Machine_Reset;
	END_IF
	IF arAxisCtrl_gb[AxisNo.TurnTable].Admin.Axis.Status.Error THEN
		arAxisCtrl_gb[AxisNo.TurnTable].Admin.ClearError := Machine_Reset;
	END_IF
	IF arAxisCtrl_gb[AxisNo.RackMotor].Admin.Axis.Status.Error THEN
		arAxisCtrl_gb[AxisNo.RackMotor].Admin.ClearError := Machine_Reset;
	END_IF
	
//////////// Cylinders
{region Cylinders }

	IF Cylinder.List.fbUpCV_FeedInPress1.xError THEN
		Cylinder.List.fbUpCV_FeedInPress1.M_Reset();
	END_IF
	IF Cylinder.List.fbUpCV_FeedInPress2.xError THEN
		Cylinder.List.fbUpCV_FeedInPress2.M_Reset();
	END_IF
	IF Cylinder.List.fbUpCV_DiameterPress.xError THEN
		Cylinder.List.fbUpCV_DiameterPress.M_Reset();
	END_IF
	IF Cylinder.List.fbUpCV_CamaraPress1.xError THEN
		Cylinder.List.fbUpCV_CamaraPress1.M_Reset();
	END_IF
	IF Cylinder.List.fbUpCV_CamaraPress2.xError THEN
		Cylinder.List.fbUpCV_CamaraPress2.M_Reset();
	END_IF
	IF Cylinder.List.fbUpCV_CamaraPress3.xError THEN
		Cylinder.List.fbUpCV_CamaraPress3.M_Reset();
	END_IF
	IF Cylinder.List.fbUpCV_CamaraPress4.xError THEN
		Cylinder.List.fbUpCV_CamaraPress4.M_Reset();
	END_IF
	IF Cylinder.List.fbUpCV_Block1.xError THEN
		Cylinder.List.fbUpCV_Block1.M_Reset();
	END_IF
	IF Cylinder.List.fbUpCV_Block2.xError THEN
		Cylinder.List.fbUpCV_Block2.M_Reset();
	END_IF
	IF Cylinder.List.fbUpCV_Block3.xError THEN
		Cylinder.List.fbUpCV_Block3.M_Reset();
	END_IF
	IF Cylinder.List.fbUpCV_DiameterHoriz.xError THEN
		Cylinder.List.fbUpCV_DiameterHoriz.M_Reset();
	END_IF
	IF Cylinder.List.fbUpCV_DiameterVert.xError THEN
		Cylinder.List.fbUpCV_DiameterVert.M_Reset();
	END_IF
	IF Cylinder.List.fbUpCV_DiameterClamp.xError THEN
		Cylinder.List.fbUpCV_DiameterClamp.M_Reset();
	END_IF
	IF Cylinder.List.fbStackPush.xError THEN
		Cylinder.List.fbStackPush.M_Reset();
	END_IF
	IF Cylinder.List.fbPullOutCV_AsidePress1.xError THEN
		Cylinder.List.fbPullOutCV_AsidePress1.M_Reset();
	END_IF
	IF Cylinder.List.fbPullOutCV_AsidePress2.xError THEN
		Cylinder.List.fbPullOutCV_AsidePress2.M_Reset();
	END_IF
	IF Cylinder.List.fbPullOutCV_AsideBlock.xError THEN
		Cylinder.List.fbPullOutCV_AsideBlock.M_Reset();
	END_IF
	IF Cylinder.List.fbPullOutCV_BsidePress1.xError THEN
		Cylinder.List.fbPullOutCV_BsidePress1.M_Reset();
	END_IF
	IF Cylinder.List.fbPullOutCV_BsidePress2.xError THEN
		Cylinder.List.fbPullOutCV_BsidePress2.M_Reset();
	END_IF
	IF Cylinder.List.fbPullOutCV_BsideBlock.xError THEN
		Cylinder.List.fbPullOutCV_BsideBlock.M_Reset();
	END_IF
	IF Cylinder.List.fbLowCV_Press1.xError THEN
		Cylinder.List.fbLowCV_Press1.M_Reset();
	END_IF
	IF Cylinder.List.fbLowCV_Press2.xError THEN
		Cylinder.List.fbLowCV_Press2.M_Reset();
	END_IF
	IF Cylinder.List.fbLowCV_Press3.xError THEN
		Cylinder.List.fbLowCV_Press3.M_Reset();
	END_IF
	IF Cylinder.List.fbLowCV_Press4.xError THEN
		Cylinder.List.fbLowCV_Press4.M_Reset();
	END_IF
	IF Cylinder.List.fbLowCV_Block1.xError THEN
		Cylinder.List.fbLowCV_Block1.M_Reset();
	END_IF
	IF Cylinder.List.fbLowCV_Block2.xError THEN
		Cylinder.List.fbLowCV_Block2.M_Reset();
	END_IF
	IF Cylinder.List.fbAllocateRobot_LeftVert1.xError THEN
		Cylinder.List.fbAllocateRobot_LeftVert1.M_Reset();
	END_IF
	IF Cylinder.List.fbAllocateRobot_LeftVert2.xError THEN
		Cylinder.List.fbAllocateRobot_LeftVert2.M_Reset();
	END_IF
	IF Cylinder.List.fbAllocateRobot_RightVert1.xError THEN
		Cylinder.List.fbAllocateRobot_RightVert1.M_Reset();
	END_IF
	IF Cylinder.List.fbAllocateRobot_RightVert2.xError THEN
		Cylinder.List.fbAllocateRobot_RightVert2.M_Reset();
	END_IF
	IF Cylinder.List.fbAllocateRobot_LeftClamp1.xError THEN
		Cylinder.List.fbAllocateRobot_LeftClamp1.M_Reset();
	END_IF
	IF Cylinder.List.fbAllocateRobot_LeftClamp2.xError THEN
		Cylinder.List.fbAllocateRobot_LeftClamp2.M_Reset();
	END_IF
	IF Cylinder.List.fbAllocateRobot_RightClamp1.xError THEN
		Cylinder.List.fbAllocateRobot_RightClamp1.M_Reset();
	END_IF
	IF Cylinder.List.fbAllocateRobot_RightClamp2.xError THEN
		Cylinder.List.fbAllocateRobot_RightClamp2.M_Reset();
	END_IF
	IF Cylinder.List.fbRoundBelt_WorkZone_Press.xError THEN
		Cylinder.List.fbRoundBelt_WorkZone_Press.M_Reset();
	END_IF
	IF Cylinder.List.fbRoundBelt_WorkZone_Plug.xError THEN
		Cylinder.List.fbRoundBelt_WorkZone_Plug.M_Reset();
	END_IF
	IF Cylinder.List.fbRoundBelt_ChargeZone_Plug.xError THEN
		Cylinder.List.fbRoundBelt_ChargeZone_Plug.M_Reset();
	END_IF
	IF Cylinder.List.fbRoundBelt_TransmitCVZone_Plug.xError THEN
		Cylinder.List.fbRoundBelt_TransmitCVZone_Plug.M_Reset();
	END_IF
	IF Cylinder.List.fbOutRobot_AsideVert.xError THEN
		Cylinder.List.fbOutRobot_AsideVert.M_Reset();
	END_IF
	IF Cylinder.List.fbOutRobot_BsideVert.xError THEN
		Cylinder.List.fbOutRobot_BsideVert.M_Reset();
	END_IF
	IF Cylinder.List.fbOutRobot_AsideClamp.xError THEN
		Cylinder.List.fbOutRobot_AsideClamp.M_Reset();
	END_IF
	IF Cylinder.List.fbOutRobot_BsideClamp.xError THEN
		Cylinder.List.fbOutRobot_BsideClamp.M_Reset();
	END_IF
	IF Cylinder.List.fbTransmitCV_CamaraHoriz.xError THEN
		Cylinder.List.fbTransmitCV_CamaraHoriz.M_Reset();
	END_IF
	IF Cylinder.List.fbDifferentSizeCV_Press2.xError THEN
		Cylinder.List.fbDifferentSizeCV_Press2.M_Reset();
	END_IF
	IF Cylinder.List.fbDifferentSizeCV_Press1.xError THEN
		Cylinder.List.fbDifferentSizeCV_Press1.M_Reset();
	END_IF
	IF Cylinder.List.fbDifferentSizeCV_Block1.xError THEN
		Cylinder.List.fbDifferentSizeCV_Block1.M_Reset();
	END_IF
	IF Cylinder.List.fbSameSizeCV_Press4.xError THEN
		Cylinder.List.fbSameSizeCV_Press4.M_Reset();
	END_IF
	IF Cylinder.List.fbSameSizeCV_Press3.xError THEN
		Cylinder.List.fbSameSizeCV_Press3.M_Reset();
	END_IF
	IF Cylinder.List.fbSameSizeCV_Press2.xError THEN
		Cylinder.List.fbSameSizeCV_Press2.M_Reset();
	END_IF
	IF Cylinder.List.fbSameSizeCV_Press1.xError THEN
		Cylinder.List.fbSameSizeCV_Press1.M_Reset();
	END_IF
	IF Cylinder.List.fbSameSizeCV_Block2.xError THEN
		Cylinder.List.fbSameSizeCV_Block2.M_Reset();
	END_IF
	IF Cylinder.List.fbSameSizeCV_Block1.xError THEN
		Cylinder.List.fbSameSizeCV_Block1.M_Reset();
	END_IF
	IF Cylinder.List.fbTurntable_Press.xError THEN
		Cylinder.List.fbTurntable_Press.M_Reset();
	END_IF
	{endregion}
	

//////////// Motor
{region Motor}
IF Motor.List.WareHouseCV_01.xError THEN
		Motor.List.WareHouseCV_01.M_Reset();
	END_IF
	IF Motor.List.WareHouseCV_02.xError THEN
		Motor.List.WareHouseCV_02.M_Reset();
	END_IF
	IF Motor.List.WareHouseCV_03.xError THEN
		Motor.List.WareHouseCV_03.M_Reset();
	END_IF
	IF Motor.List.WareHouseCV_04.xError THEN
		Motor.List.WareHouseCV_04.M_Reset();
	END_IF
	IF Motor.List.WareHouseCV_05.xError THEN
		Motor.List.WareHouseCV_05.M_Reset();
	END_IF
	IF Motor.List.WareHouseCV_06.xError THEN
		Motor.List.WareHouseCV_06.M_Reset();
	END_IF
	IF Motor.List.WareHouseCV_07.xError THEN
		Motor.List.WareHouseCV_07.M_Reset();
	END_IF
	IF Motor.List.WareHouseCV_08.xError THEN
		Motor.List.WareHouseCV_08.M_Reset();
	END_IF
	IF Motor.List.WareHouseCV_09.xError THEN
		Motor.List.WareHouseCV_09.M_Reset();
	END_IF
	IF Motor.List.WareHouseCV_10.xError THEN
		Motor.List.WareHouseCV_10.M_Reset();
	END_IF
	IF Motor.List.WareHouseCV_11.xError THEN
		Motor.List.WareHouseCV_11.M_Reset();
	END_IF
	IF Motor.List.WareHouseCV_12.xError THEN
		Motor.List.WareHouseCV_12.M_Reset();
	END_IF
	IF Motor.List.WareHouseCV_13.xError THEN
		Motor.List.WareHouseCV_13.M_Reset();
	END_IF
	IF Motor.List.WareHouseCV_14.xError THEN
		Motor.List.WareHouseCV_14.M_Reset();
	END_IF
	IF Motor.List.WareHouseCV_15.xError THEN
		Motor.List.WareHouseCV_15.M_Reset();
	END_IF
	IF Motor.List.WareHouseCV_16.xError THEN
		Motor.List.WareHouseCV_16.M_Reset();
	END_IF
	IF Motor.List.WareHouseCV_17.xError THEN
		Motor.List.WareHouseCV_17.M_Reset();
	END_IF
	IF Motor.List.WareHouseCV_18.xError THEN
		Motor.List.WareHouseCV_18.M_Reset();
	END_IF
	IF Motor.List.WareHouseCV_19.xError THEN
		Motor.List.WareHouseCV_19.M_Reset();
	END_IF
	IF Motor.List.WareHouseCV_20.xError THEN
		Motor.List.WareHouseCV_20.M_Reset();
	END_IF
	IF Motor.List.UpCV.xError THEN
		Motor.List.UpCV.M_Reset();
	END_IF
	IF Motor.List.LowCV.xError THEN
		Motor.List.LowCV.M_Reset();
	END_IF
	IF Motor.List.PullOutCV_A.xError THEN
		Motor.List.PullOutCV_A.M_Reset();
	END_IF
	IF Motor.List.PullOutCV_B.xError THEN
		Motor.List.PullOutCV_B.M_Reset();
	END_IF
	IF Motor.List.TransmitSameSideCV.xError THEN
		Motor.List.TransmitSameSideCV.M_Reset();
	END_IF
	IF Motor.List.TransmitDifferentSideCV.xError THEN
		Motor.List.TransmitDifferentSideCV.M_Reset();
	END_IF	 
{endregion}
	SafeDoorResetError := TRUE;		//Edited by Gamin 2025/11/22


ELSIF ResetEdgeDetect.xFallingEdge THEN
	arAxisCtrl_gb[AxisNo.Allocate_X].Admin.ClearError := Machine_Reset;
	arAxisCtrl_gb[AxisNo.Allocate_Y].Admin.ClearError := Machine_Reset;
	arAxisCtrl_gb[AxisNo.OutRobot_X].Admin.ClearError := Machine_Reset;
	arAxisCtrl_gb[AxisNo.OutRobot_Y].Admin.ClearError := Machine_Reset;
	arAxisCtrl_gb[AxisNo.RoundBelt].Admin.ClearError := Machine_Reset;
	arAxisCtrl_gb[AxisNo.TurnTable].Admin.ClearError := Machine_Reset;
	arAxisCtrl_gb[AxisNo.RackMotor].Admin.ClearError := Machine_Reset;
	SafeDoorResetError := FALSE;	//Cleared residual TRUE flags
END_IF

IF SafeDoorResetError THEN
	FOR i := 1 TO 20 DO 
		SafeDoorsOpen[i] := FALSE;
	END_FOR
END_IF

Error := xError;
ErrorID := xErrorID;
ErrMsg := xErrorMsg;
END_ACTION

ACTION A20_ConveyorArbitration:
// 同尺寸軌道集中式仲裁 (Phase 2)
// 取各 sub-FB 的請求 flag 做 OR,優先序:HoldStill > 方向衝突 (停) > Backward > Forward > 預設停。
// Sub-FB 不再直接 call M_MoveBackward / M_MotorStop。

// 手動模式 yield:MotorManualCtrl[25] 在 manual 命令按下時負責驅動 motor,A20 不干涉避免 M_MotorStop 蓋掉 manual。
IF AllocateManualCommand.TransCV.TransmitSameSideCV.Forward
   OR AllocateManualCommand.TransCV.TransmitSameSideCV.Backward
   OR AllocateManualCommand.TransCV.TransmitSameSideCV.Stopped THEN
	RETURN;
END_IF

IF SameSizeCVRequest.bCamera_HoldStill OR SameSizeCVRequest.bWareHouse_HoldStill THEN
	// 任何 sub-FB 要靜止 (拍照 / 取盒對位) — 強制停
	Motor.List.TransmitSameSideCV.M_MotorStop();
ELSIF (SameSizeCVRequest.bScan_NeedBackward
       OR SameSizeCVRequest.bShippingTransfer_NeedBackward
       OR SameSizeCVRequest.bCamera_NeedBackward
       OR SameSizeCVRequest.bWareHouse_NeedBackward)
      AND SameSizeCVRequest.bShippingTransfer_NeedForward THEN
	// 方向衝突 (不應該發生) — 安全起見停下,讓 sub-FB 自己解
	Motor.List.TransmitSameSideCV.M_MotorStop();
ELSIF SameSizeCVRequest.bScan_NeedBackward
      OR SameSizeCVRequest.bShippingTransfer_NeedBackward
      OR SameSizeCVRequest.bCamera_NeedBackward
      OR SameSizeCVRequest.bWareHouse_NeedBackward THEN
	IF NOT Motor.List.TransmitSameSideCV.InForWard THEN
		Motor.List.TransmitSameSideCV.M_MoveBackward();
	END_IF
ELSIF SameSizeCVRequest.bShippingTransfer_NeedForward THEN
	IF NOT Motor.List.TransmitSameSideCV.InBackWard THEN
		Motor.List.TransmitSameSideCV.M_MoveForward();
	END_IF
ELSE
	// 沒人要 → 停 (例:本批做完所有 sub-FB 進 DONE,flag 自動清)
	Motor.List.TransmitSameSideCV.M_MotorStop();
END_IF
END_ACTION

METHOD M_Aborted
VAR
	CylinderIndex :UDINT;
	MotorIndex : INT;
	ServoIndex : INT;
END_VAR
IF eModeCommand = E_UnitMode.Auto THEN
    GVL_Machine.PackTags[UnitNo.Storage].Command.UnitMode := E_UnitMode.Auto;
    GVL_Machine.PackTags[UnitNo.Allocate].Command.UnitMode := E_UnitMode.Auto;
    GVL_Machine.PackTags[UnitNo.Shipping].Command.UnitMode := E_UnitMode.Auto;
ELSIF eModeCommand = E_UnitMode.Manual THEN
    GVL_Machine.PackTags[UnitNo.Storage].Command.UnitMode := E_UnitMode.Manual;
    GVL_Machine.PackTags[UnitNo.Allocate].Command.UnitMode := E_UnitMode.Manual;
    GVL_Machine.PackTags[UnitNo.Shipping].Command.UnitMode := E_UnitMode.Manual;
END_IF

FOR ServoIndex := 1 TO 7 DO
    arAxisCtrl_gb[ServoIndex].Admin._OpMode.en := ModeAH;
END_FOR

CASE eModeCurrent OF
    E_UnitMode.Manual:
        IF GVL_Machine.PackTags[UnitNo.Allocate].Status.UnitModeCurrent = E_UnitMode.Manual AND
            GVL_Machine.PackTags[UnitNo.Allocate].Status.StateCurrent = ePMLState_Aborted AND
            GVL_Machine.PackTags[UnitNo.Storage].Status.UnitModeCurrent = E_UnitMode.Manual AND
            GVL_Machine.PackTags[UnitNo.Storage].Status.StateCurrent = ePMLState_Aborted AND
            GVL_Machine.PackTags[UnitNo.Shipping].Status.UnitModeCurrent = E_UnitMode.Manual AND
            GVL_Machine.PackTags[UnitNo.Shipping].Status.StateCurrent = ePMLState_Aborted THEN
            IF NOT Error OR Machine_Reset THEN
                M_StateComplete();
            END_IF
        END_IF
    E_UnitMode.Auto:
        IF GVL_Machine.PackTags[UnitNo.Allocate].Status.UnitModeCurrent = E_UnitMode.Auto AND
            GVL_Machine.PackTags[UnitNo.Allocate].Status.StateCurrent = ePMLState_Aborted AND
            GVL_Machine.PackTags[UnitNo.Storage].Status.UnitModeCurrent = E_UnitMode.Auto AND
            GVL_Machine.PackTags[UnitNo.Storage].Status.StateCurrent = ePMLState_Aborted AND
            GVL_Machine.PackTags[UnitNo.Shipping].Status.UnitModeCurrent = E_UnitMode.Auto AND
            GVL_Machine.PackTags[UnitNo.Shipping].Status.StateCurrent = ePMLState_Aborted THEN
            IF NOT Error OR Machine_Reset THEN
                M_StateComplete();
            END_IF
        END_IF
END_CASE
END_METHOD

METHOD M_Aborting
VAR
	CylinderIndex :UDINT;
	MotorIndex : INT;
	ServoIndex : INT;
END_VAR
CASE eModeCurrent OF
    E_UnitMode.Manual:
        GVL_Machine.PackTags[UnitNo.Allocate].Command.UnitMode := E_UnitMode.Manual;
        GVL_Machine.PackTags[UnitNo.Allocate].Command.CntrlCmd := ePMLCommand_Abort;
        GVL_Machine.PackTags[UnitNo.Storage].Command.UnitMode  := E_UnitMode.Manual;
        GVL_Machine.PackTags[UnitNo.Storage].Command.CntrlCmd  := ePMLCommand_Abort;
        GVL_Machine.PackTags[UnitNo.Shipping].Command.UnitMode := E_UnitMode.Manual;
        GVL_Machine.PackTags[UnitNo.Shipping].Command.CntrlCmd := ePMLCommand_Abort;
		FOR CylinderIndex := 1 TO udiMax_CylinderNum DO
			Cylinder.arCylinder[CylinderIndex].xEnable := FALSE;
		END_FOR
		FOR MotorIndex := 1 TO 26 DO
			Motor.arMotor[MotorIndex].xEnable := FALSE;
		END_FOR
		TableMove.xExecute := FALSE;
        IF GVL_Machine.PackTags[UnitNo.Allocate].Status.UnitModeCurrent = E_UnitMode.Manual AND
           GVL_Machine.PackTags[UnitNo.Allocate].Status.StateCurrent = ePMLState_Aborting AND
           GVL_Machine.PackTags[UnitNo.Storage].Status.UnitModeCurrent = E_UnitMode.Manual AND
           GVL_Machine.PackTags[UnitNo.Storage].Status.StateCurrent = ePMLState_Aborting AND
           GVL_Machine.PackTags[UnitNo.Shipping].Status.UnitModeCurrent = E_UnitMode.Manual AND
           GVL_Machine.PackTags[UnitNo.Shipping].Status.StateCurrent = ePMLState_Aborting AND NOT
		   TableMove.xError
            THEN
            M_StateComplete();
        END_IF
	E_UnitMode.Auto:
        GVL_Machine.PackTags[UnitNo.Allocate].Command.UnitMode := E_UnitMode.Auto;
        GVL_Machine.PackTags[UnitNo.Allocate].Command.CntrlCmd := ePMLCommand_Abort;
        GVL_Machine.PackTags[UnitNo.Storage].Command.UnitMode  := E_UnitMode.Auto;
        GVL_Machine.PackTags[UnitNo.Storage].Command.CntrlCmd  := ePMLCommand_Abort;
        GVL_Machine.PackTags[UnitNo.Shipping].Command.UnitMode := E_UnitMode.Auto;
        GVL_Machine.PackTags[UnitNo.Shipping].Command.CntrlCmd := ePMLCommand_Abort;
		FOR CylinderIndex := 1 TO udiMax_CylinderNum DO
			Cylinder.arCylinder[CylinderIndex].xEnable := FALSE;
		END_FOR
		FOR MotorIndex := 1 TO 26 DO
			Motor.arMotor[MotorIndex].xEnable := FALSE;
		END_FOR
		TableMove.xExecute := FALSE;
        IF GVL_Machine.PackTags[UnitNo.Allocate].Status.UnitModeCurrent = E_UnitMode.Auto AND
           GVL_Machine.PackTags[UnitNo.Allocate].Status.StateCurrent = ePMLState_Aborting AND
           GVL_Machine.PackTags[UnitNo.Storage].Status.UnitModeCurrent = E_UnitMode.Auto AND
           GVL_Machine.PackTags[UnitNo.Storage].Status.StateCurrent = ePMLState_Aborting AND
           GVL_Machine.PackTags[UnitNo.Shipping].Status.UnitModeCurrent = E_UnitMode.Auto AND
           GVL_Machine.PackTags[UnitNo.Shipping].Status.StateCurrent = ePMLState_Aborting AND NOT
		   TableMove.xError
            THEN
            M_StateComplete();
        END_IF
END_CASE
FOR ServoIndex:=1 TO 7 DO
	arAxisCtrl_gb[ServoIndex].Admin._OpMode.en := ModeAH;
END_FOR
END_METHOD

METHOD PRIVATE M_Auto_Axes : BOOL
VAR_INPUT
END_VAR

VAR_INST
	AllowAllocateRobotMove : BOOL;
	AllowOutRobotMove : BOOL;
	AllowRoundBeltMove : BOOL;
	AllowTurnTable		:BOOL;
	AllowRackMotor		:BOOL;
END_VAR
// Safe check
AllowAllocateRobotMove := Cylinder.List.fbAllocateRobot_LeftVert1.InRearPosition AND
    Cylinder.List.fbAllocateRobot_LeftVert2.InRearPosition AND
    Cylinder.List.fbAllocateRobot_RightVert1.InRearPosition AND
    Cylinder.List.fbAllocateRobot_RightVert2.InRearPosition;

AllowOutRobotMove := Cylinder.List.fbOutRobot_AsideVert.InRearPosition AND Cylinder.List.fbOutRobot_BsideVert.InRearPosition;
AllowRoundBeltMove := Cylinder.List.fbRoundBelt_ChargeZone_Plug.InRearPosition AND
    Cylinder.List.fbRoundBelt_TransmitCVZone_Plug.InRearPosition AND
    Cylinder.List.fbRoundBelt_WorkZone_Plug.InRearPosition AND
    Cylinder.List.fbRoundBelt_WorkZone_Press.InRearPosition AND
    AllowAllocateRobotMove AND
    AllowOutRobotMove
	AND NOT FanucRobot.List.StorageRobot.BZoneInWork AND NOT FanucRobot.List.StorageRobot.Bzone_AllowWork;;

AllowTurnTable := Cylinder.List.fbTurntable_Press.InRearPosition;
AllowRackMotor := Cylinder.List.fbStackPush.InRearPosition;

// Axis controll
{region "AllocateRobot AxisX"}

IF AllocateManualCommand.AllocatedRobot.AxisX.JOG.MoveFWD AND AllowAllocateRobotMove THEN
    arAxisCtrl_gb[AxisNo.Allocate_X].VelMode.Acc := CurrentData.Axes.Allocate_X.Manual.JogAcceleration;
    arAxisCtrl_gb[AxisNo.Allocate_X].VelMode.Dec := CurrentData.Axes.Allocate_X.Manual.JogDeceleration;
    arAxisCtrl_gb[AxisNo.Allocate_X].VelMode.Jerk := CurrentData.Axes.Allocate_X.Manual.JogJerk;
    arAxisCtrl_gb[AxisNo.Allocate_X].VelMode.Velocity := CurrentData.Axes.Allocate_X.Manual.JogVelocity;
    arAxisCtrl_gb[AxisNo.Allocate_X].Admin._OpMode.en := E_AXIS_MODE.ModeVel;
ELSIF AllocateManualCommand.AllocatedRobot.AxisX.JOG.MoveBWD AND AllowAllocateRobotMove THEN
    arAxisCtrl_gb[AxisNo.Allocate_X].VelMode.Acc := CurrentData.Axes.Allocate_X.Manual.JogAcceleration;
    arAxisCtrl_gb[AxisNo.Allocate_X].VelMode.Dec := CurrentData.Axes.Allocate_X.Manual.JogDeceleration;
    arAxisCtrl_gb[AxisNo.Allocate_X].VelMode.Jerk := CurrentData.Axes.Allocate_X.Manual.JogJerk;
    arAxisCtrl_gb[AxisNo.Allocate_X].VelMode.Velocity := CurrentData.Axes.Allocate_X.Manual.JogVelocity * -1;
    arAxisCtrl_gb[AxisNo.Allocate_X].Admin._OpMode.en := E_AXIS_MODE.ModeVel;
ELSIF AllocateManualCommand.AllocatedRobot.AxisX.PTP.Enable AND AllowAllocateRobotMove THEN
    arAxisCtrl_gb[AxisNo.Allocate_X].PosMode.Acc := CurrentData.Axes.Allocate_X.Manual.PtpAcceleration;
    arAxisCtrl_gb[AxisNo.Allocate_X].PosMode.Dec := CurrentData.Axes.Allocate_X.Manual.PtpDeceleration;
    arAxisCtrl_gb[AxisNo.Allocate_X].PosMode.Jerk := CurrentData.Axes.Allocate_X.Manual.PtpJerk;
    arAxisCtrl_gb[AxisNo.Allocate_X].PosMode.Velocity := CurrentData.Axes.Allocate_X.Manual.PtpVelocity;
    arAxisCtrl_gb[AxisNo.Allocate_X].PosMode.Position := CurrentData.Axes.Allocate_X.Manual.PtpPosition;
    arAxisCtrl_gb[AxisNo.Allocate_X].Admin._OpMode.en := ModePosAbs;
ELSIF (AllocateManualCommand.AllocatedRobot.AxisX.Homing.Execute OR  fbAllocateArea.fbAllocateHome.AxisHomingRequest)  AND AllowAllocateRobotMove THEN
    arAxisCtrl_gb[AxisNo.Allocate_X].SetupMode.eHomingMode := E_HomingMode._17_Neg_LimitOutterRight;
    arAxisCtrl_gb[AxisNo.Allocate_X].SetupMode.FastVelo := CurrentData.Axes.Allocate_X.Homing.FastVelo;
    arAxisCtrl_gb[AxisNo.Allocate_X].SetupMode.SlowVelo := CurrentData.Axes.Allocate_X.Homing.SlowVelo;
    arAxisCtrl_gb[AxisNo.Allocate_X].SetupMode.lrOffset := CurrentData.Axes.Allocate_X.Homing.Offset;
    arAxisCtrl_gb[AxisNo.Allocate_X].SetupMode.lrSetPosition := CurrentData.Axes.Allocate_X.Homing.SetAbsolutePosition;
    arAxisCtrl_gb[AxisNo.Allocate_X].SetupMode.stPosBiasParameter.bSetPostionBias := TRUE;
    arAxisCtrl_gb[AxisNo.Allocate_X].Admin._OpMode.en := ModeHoming;
ELSIF TableMove.xBusy AND AllowAllocateRobotMove THEN
    arAxisCtrl_gb[AxisNo.Allocate_X].Admin._OpMode.en := ModePosAbs;
ELSIF fbAllocateArea.fb_AllocateBatchMode.Busy AND AllowAllocateRobotMove THEN
    arAxisCtrl_gb[AxisNo.Allocate_X].Admin._OpMode.en := ModePosAbs;
ELSIF fbAllocateArea.fb_AllocateBatchMode_Reverse.Busy AND fbAllocateArea.fb_AllocateBatchMode_Reverse.bAllocateRobotMoveRequest AND AllowAllocateRobotMove THEN
	arAxisCtrl_gb[AxisNo.Allocate_X].Admin._OpMode.en := ModePosAbs;
ELSE
    arAxisCtrl_gb[AxisNo.Allocate_X].Admin.StopDeceleration := 1000;
    arAxisCtrl_gb[AxisNo.Allocate_X].Admin._OpMode.en := E_AXIS_MODE.ModeAH;
		 
END_IF
{endregion}

{region "AllocateRobot AxisY"}
IF AllocateManualCommand.AllocatedRobot.AxisY.JOG.MoveFWD AND AllowAllocateRobotMove THEN
    arAxisCtrl_gb[AxisNo.Allocate_Y].VelMode.Acc := CurrentData.Axes.Allocate_Y.Manual.JogAcceleration;
    arAxisCtrl_gb[AxisNo.Allocate_Y].VelMode.Dec := CurrentData.Axes.Allocate_Y.Manual.JogDeceleration;
    arAxisCtrl_gb[AxisNo.Allocate_Y].VelMode.Jerk := CurrentData.Axes.Allocate_Y.Manual.JogJerk;
    arAxisCtrl_gb[AxisNo.Allocate_Y].VelMode.Velocity := CurrentData.Axes.Allocate_Y.Manual.JogVelocity;
    arAxisCtrl_gb[AxisNo.Allocate_Y].Admin._OpMode.en := E_AXIS_MODE.ModeVel;
ELSIF AllocateManualCommand.AllocatedRobot.AxisY.JOG.MoveBWD AND AllowAllocateRobotMove THEN
    arAxisCtrl_gb[AxisNo.Allocate_Y].VelMode.Acc := CurrentData.Axes.Allocate_Y.Manual.JogAcceleration;
    arAxisCtrl_gb[AxisNo.Allocate_Y].VelMode.Dec := CurrentData.Axes.Allocate_Y.Manual.JogDeceleration;
    arAxisCtrl_gb[AxisNo.Allocate_Y].VelMode.Jerk := CurrentData.Axes.Allocate_Y.Manual.JogJerk;
    arAxisCtrl_gb[AxisNo.Allocate_Y].VelMode.Velocity := CurrentData.Axes.Allocate_Y.Manual.JogVelocity * -1;
    arAxisCtrl_gb[AxisNo.Allocate_Y].Admin._OpMode.en := E_AXIS_MODE.ModeVel;
ELSIF AllocateManualCommand.AllocatedRobot.AxisY.PTP.Enable AND AllowAllocateRobotMove THEN
    arAxisCtrl_gb[AxisNo.Allocate_Y].PosMode.Acc := CurrentData.Axes.Allocate_Y.Manual.PtpAcceleration;
    arAxisCtrl_gb[AxisNo.Allocate_Y].PosMode.Dec := CurrentData.Axes.Allocate_Y.Manual.PtpDeceleration;
    arAxisCtrl_gb[AxisNo.Allocate_Y].PosMode.Jerk := CurrentData.Axes.Allocate_Y.Manual.PtpJerk;
    arAxisCtrl_gb[AxisNo.Allocate_Y].PosMode.Velocity := CurrentData.Axes.Allocate_Y.Manual.PtpVelocity;
    arAxisCtrl_gb[AxisNo.Allocate_Y].PosMode.Position := CurrentData.Axes.Allocate_Y.Manual.PtpPosition;
    arAxisCtrl_gb[AxisNo.Allocate_Y].Admin._OpMode.en := ModePosAbs;
//ELSIF( AllocateManualCommand.AllocatedRobot.AxisY.Homing.Execute OR  fbAllocateArea.fbAllocateHome.AxisHomingRequest ) AND AllowAllocateRobotMove THEN
//    arAxisCtrl_gb[AxisNo.Allocate_Y].SetupMode.eHomingMode := E_HomingMode._36_MoveToAbsHomePoint;
//    arAxisCtrl_gb[AxisNo.Allocate_Y].SetupMode.FastVelo := CurrentData.Axes.Allocate_Y.Homing.FastVelo;
//    arAxisCtrl_gb[AxisNo.Allocate_Y].SetupMode.SlowVelo := CurrentData.Axes.Allocate_Y.Homing.SlowVelo;
//    arAxisCtrl_gb[AxisNo.Allocate_Y].SetupMode.lrOffset := CurrentData.Axes.Allocate_Y.Homing.Offset;
//    arAxisCtrl_gb[AxisNo.Allocate_Y].SetupMode.lrSetPosition := CurrentData.Axes.Allocate_Y.Homing.SetAbsolutePosition;
//    arAxisCtrl_gb[AxisNo.Allocate_Y].SetupMode.stPosBiasParameter.bSetPostionBias := FALSE;
//    arAxisCtrl_gb[AxisNo.Allocate_Y].Admin._OpMode.en := ModeHoming;
ELSIF( AllocateManualCommand.AllocatedRobot.AxisY.Homing.Execute OR  fbAllocateArea.fbAllocateHome.AxisHomingRequest ) AND AllowAllocateRobotMove THEN
    arAxisCtrl_gb[AxisNo.Allocate_Y].PosMode.Acc := CurrentData.Axes.Allocate_Y.Homing.FastVelo.Acc;
    arAxisCtrl_gb[AxisNo.Allocate_Y].PosMode.Dec := CurrentData.Axes.Allocate_Y.Homing.FastVelo.Dec;
    arAxisCtrl_gb[AxisNo.Allocate_Y].PosMode.Jerk := CurrentData.Axes.Allocate_Y.Homing.FastVelo.Jerk;
    arAxisCtrl_gb[AxisNo.Allocate_Y].PosMode.Velocity := CurrentData.Axes.Allocate_Y.Homing.FastVelo.Velocity;
    arAxisCtrl_gb[AxisNo.Allocate_Y].PosMode.Position := CurrentData.Axes.Allocate_Y.Homing.Offset;
    arAxisCtrl_gb[AxisNo.Allocate_Y].Admin._OpMode.en := ModePosAbs;
		 
    IF arAxisStatus_gb[AxisNo.Allocate_Y].Admin._OpModeAck = ModePosAbs AND arAxisStatus_gb[AxisNo.Allocate_Y].Admin.CmdDone THEN
        GVL_Machine.AllocatYAxisHome := TRUE;
    END_IF
ELSIF TableMove.xBusy AND AllowAllocateRobotMove THEN
    arAxisCtrl_gb[AxisNo.Allocate_Y].Admin._OpMode.en := ModePosAbs;
ELSIF fbAllocateArea.fb_AllocateBatchMode.Busy AND AllowAllocateRobotMove THEN
    arAxisCtrl_gb[AxisNo.Allocate_Y].Admin._OpMode.en := ModePosAbs;
ELSIF fbAllocateArea.fb_AllocateBatchMode_Reverse.Busy AND fbAllocateArea.fb_AllocateBatchMode_Reverse.bAllocateRobotMoveRequest AND AllowAllocateRobotMove THEN
	arAxisCtrl_gb[AxisNo.Allocate_Y].Admin._OpMode.en := ModePosAbs;
ELSE
    arAxisCtrl_gb[AxisNo.Allocate_Y].Admin.StopDeceleration := 1000;
    arAxisCtrl_gb[AxisNo.Allocate_Y].Admin._OpMode.en := E_AXIS_MODE.ModeAH;
END_IF

{EndRegion}

{region "OutRobot AxisX"}
IF AllocateManualCommand.OutRobot.AxisX.JOG.MoveFWD AND AllowOutRobotMove THEN
    arAxisCtrl_gb[AxisNo.OutRobot_X].VelMode.Acc := CurrentData.Axes.OutRobot_X.Manual.JogAcceleration;
    arAxisCtrl_gb[AxisNo.OutRobot_X].VelMode.Dec := CurrentData.Axes.OutRobot_X.Manual.JogDeceleration;
    arAxisCtrl_gb[AxisNo.OutRobot_X].VelMode.Jerk := CurrentData.Axes.OutRobot_X.Manual.JogJerk;
    arAxisCtrl_gb[AxisNo.OutRobot_X].VelMode.Velocity := CurrentData.Axes.OutRobot_X.Manual.JogVelocity;
    arAxisCtrl_gb[AxisNo.OutRobot_X].Admin._OpMode.en := E_AXIS_MODE.ModeVel;
ELSIF AllocateManualCommand.OutRobot.AxisX.JOG.MoveBWD AND AllowOutRobotMove THEN
    arAxisCtrl_gb[AxisNo.OutRobot_X].VelMode.Acc := CurrentData.Axes.OutRobot_X.Manual.JogAcceleration;
    arAxisCtrl_gb[AxisNo.OutRobot_X].VelMode.Dec := CurrentData.Axes.OutRobot_X.Manual.JogDeceleration;
    arAxisCtrl_gb[AxisNo.OutRobot_X].VelMode.Jerk := CurrentData.Axes.OutRobot_X.Manual.JogJerk;
    arAxisCtrl_gb[AxisNo.OutRobot_X].VelMode.Velocity := CurrentData.Axes.OutRobot_X.Manual.JogVelocity * -1;
    arAxisCtrl_gb[AxisNo.OutRobot_X].Admin._OpMode.en := E_AXIS_MODE.ModeVel;
ELSIF AllocateManualCommand.OutRobot.AxisX.PTP.Enable AND AllowOutRobotMove THEN
    arAxisCtrl_gb[AxisNo.OutRobot_X].PosMode.Acc := CurrentData.Axes.OutRobot_X.Manual.PtpAcceleration;
    arAxisCtrl_gb[AxisNo.OutRobot_X].PosMode.Dec := CurrentData.Axes.OutRobot_X.Manual.PtpDeceleration;
    arAxisCtrl_gb[AxisNo.OutRobot_X].PosMode.Jerk := CurrentData.Axes.OutRobot_X.Manual.PtpJerk;
    arAxisCtrl_gb[AxisNo.OutRobot_X].PosMode.Velocity := CurrentData.Axes.OutRobot_X.Manual.PtpVelocity;
    arAxisCtrl_gb[AxisNo.OutRobot_X].PosMode.Position := CurrentData.Axes.OutRobot_X.Manual.PtpPosition;
    arAxisCtrl_gb[AxisNo.OutRobot_X].Admin._OpMode.en := ModePosAbs;
ELSIF (AllocateManualCommand.OutRobot.AxisX.Homing.Execute OR  fbAllocateArea.fbAllocateHome.AxisHomingRequest ) AND AllowOutRobotMove THEN
    arAxisCtrl_gb[AxisNo.OutRobot_X].SetupMode.eHomingMode := E_HomingMode._28_Neg_HomeInnerRight_withLimit;
    arAxisCtrl_gb[AxisNo.OutRobot_X].SetupMode.FastVelo := CurrentData.Axes.OutRobot_X.Homing.FastVelo;
    arAxisCtrl_gb[AxisNo.OutRobot_X].SetupMode.SlowVelo := CurrentData.Axes.OutRobot_X.Homing.SlowVelo;
    arAxisCtrl_gb[AxisNo.OutRobot_X].SetupMode.lrOffset := CurrentData.Axes.OutRobot_X.Homing.Offset;
    arAxisCtrl_gb[AxisNo.OutRobot_X].SetupMode.lrSetPosition := CurrentData.Axes.OutRobot_X.Homing.SetAbsolutePosition;
    arAxisCtrl_gb[AxisNo.OutRobot_X].SetupMode.stPosBiasParameter.bSetPostionBias := TRUE;
    arAxisCtrl_gb[AxisNo.OutRobot_X].Admin._OpMode.en := ModeHoming;
ELSIF TableMove.xBusy AND AllowOutRobotMove THEN
	arAxisCtrl_gb[AxisNo.OutRobot_X].PosMode.Acc := CurrentData.Axes.OutRobot_X.HalfAuto.Acceleration;
    arAxisCtrl_gb[AxisNo.OutRobot_X].PosMode.Dec := CurrentData.Axes.OutRobot_X.HalfAuto.Deceleration;
    arAxisCtrl_gb[AxisNo.OutRobot_X].PosMode.Jerk := CurrentData.Axes.OutRobot_X.HalfAuto.Jerk;
    arAxisCtrl_gb[AxisNo.OutRobot_X].PosMode.Velocity := CurrentData.Axes.OutRobot_X.HalfAuto.Velocity;		   
    arAxisCtrl_gb[AxisNo.OutRobot_X].Admin._OpMode.en := ModePosAbs;
ELSIF (AllocateService.AutoMode_BoxMoveReverse.HandShake.Busy 
	  OR AllocateService.AutoMode_EmptyBoxMove.HandShake.Busy 
	  OR AllocateService.AutoMode_RareBoxMove.HandShake.Busy) AND AllowOutRobotMove THEN
	arAxisCtrl_gb[AxisNo.OutRobot_X].PosMode.Acc := CurrentData.Axes.OutRobot_X.Auto.Acceleration;
    arAxisCtrl_gb[AxisNo.OutRobot_X].PosMode.Dec := CurrentData.Axes.OutRobot_X.Auto.Deceleration;
    arAxisCtrl_gb[AxisNo.OutRobot_X].PosMode.Jerk := CurrentData.Axes.OutRobot_X.Auto.Jerk;
    arAxisCtrl_gb[AxisNo.OutRobot_X].PosMode.Velocity := CurrentData.Axes.OutRobot_X.Auto.Velocity;		   
    arAxisCtrl_gb[AxisNo.OutRobot_X].Admin._OpMode.en := ModePosAbs;
ELSE
    arAxisCtrl_gb[AxisNo.OutRobot_X].Admin.StopDeceleration := 1000;
    arAxisCtrl_gb[AxisNo.OutRobot_X].Admin._OpMode.en := E_AXIS_MODE.ModeAH;
END_IF

{Endregion}

{region "OutRobot AxisY"}
IF AllocateManualCommand.OutRobot.AxisY.JOG.MoveFWD AND AllowOutRobotMove THEN
    arAxisCtrl_gb[AxisNo.OutRobot_Y].VelMode.Acc := CurrentData.Axes.OutRobot_Y.Manual.JogAcceleration;
    arAxisCtrl_gb[AxisNo.OutRobot_Y].VelMode.Dec := CurrentData.Axes.OutRobot_Y.Manual.JogDeceleration;
    arAxisCtrl_gb[AxisNo.OutRobot_Y].VelMode.Jerk := CurrentData.Axes.OutRobot_Y.Manual.JogJerk;
    arAxisCtrl_gb[AxisNo.OutRobot_Y].VelMode.Velocity := CurrentData.Axes.OutRobot_Y.Manual.JogVelocity;
    arAxisCtrl_gb[AxisNo.OutRobot_Y].Admin._OpMode.en := E_AXIS_MODE.ModeVel;
ELSIF AllocateManualCommand.OutRobot.AxisY.JOG.MoveBWD AND AllowOutRobotMove THEN
    arAxisCtrl_gb[AxisNo.OutRobot_Y].VelMode.Acc := CurrentData.Axes.OutRobot_Y.Manual.JogAcceleration;
    arAxisCtrl_gb[AxisNo.OutRobot_Y].VelMode.Dec := CurrentData.Axes.OutRobot_Y.Manual.JogDeceleration;
    arAxisCtrl_gb[AxisNo.OutRobot_Y].VelMode.Jerk := CurrentData.Axes.OutRobot_Y.Manual.JogJerk;
    arAxisCtrl_gb[AxisNo.OutRobot_Y].VelMode.Velocity := CurrentData.Axes.OutRobot_Y.Manual.JogVelocity * -1;
    arAxisCtrl_gb[AxisNo.OutRobot_Y].Admin._OpMode.en := E_AXIS_MODE.ModeVel;
ELSIF AllocateManualCommand.OutRobot.AxisY.PTP.Enable AND AllowOutRobotMove THEN
    arAxisCtrl_gb[AxisNo.OutRobot_Y].PosMode.Acc := CurrentData.Axes.OutRobot_Y.Manual.PtpAcceleration;
    arAxisCtrl_gb[AxisNo.OutRobot_Y].PosMode.Dec := CurrentData.Axes.OutRobot_Y.Manual.PtpDeceleration;
    arAxisCtrl_gb[AxisNo.OutRobot_Y].PosMode.Jerk := CurrentData.Axes.OutRobot_Y.Manual.PtpJerk;
    arAxisCtrl_gb[AxisNo.OutRobot_Y].PosMode.Velocity := CurrentData.Axes.OutRobot_Y.Manual.PtpVelocity;
    arAxisCtrl_gb[AxisNo.OutRobot_Y].PosMode.Position := CurrentData.Axes.OutRobot_Y.Manual.PtpPosition;
    arAxisCtrl_gb[AxisNo.OutRobot_Y].Admin._OpMode.en := ModePosAbs;
ELSIF (AllocateManualCommand.OutRobot.AxisY.Homing.Execute OR  fbAllocateArea.fbAllocateHome.AxisHomingRequest) AND AllowOutRobotMove THEN
    arAxisCtrl_gb[AxisNo.OutRobot_Y].SetupMode.eHomingMode := E_HomingMode._28_Neg_HomeInnerRight_withLimit;
    arAxisCtrl_gb[AxisNo.OutRobot_Y].SetupMode.FastVelo := CurrentData.Axes.OutRobot_Y.Homing.FastVelo;
    arAxisCtrl_gb[AxisNo.OutRobot_Y].SetupMode.SlowVelo := CurrentData.Axes.OutRobot_Y.Homing.SlowVelo;
    arAxisCtrl_gb[AxisNo.OutRobot_Y].SetupMode.lrOffset := CurrentData.Axes.OutRobot_Y.Homing.Offset;
    arAxisCtrl_gb[AxisNo.OutRobot_Y].SetupMode.lrSetPosition := CurrentData.Axes.OutRobot_Y.Homing.SetAbsolutePosition;
    arAxisCtrl_gb[AxisNo.OutRobot_Y].SetupMode.stPosBiasParameter.bSetPostionBias := TRUE;
    arAxisCtrl_gb[AxisNo.OutRobot_Y].Admin._OpMode.en := ModeHoming;
ELSIF TableMove.xBusy AND AllowOutRobotMove THEN
	arAxisCtrl_gb[AxisNo.OutRobot_Y].PosMode.Acc := CurrentData.Axes.OutRobot_Y.HalfAuto.Acceleration;
    arAxisCtrl_gb[AxisNo.OutRobot_Y].PosMode.Dec := CurrentData.Axes.OutRobot_Y.HalfAuto.Deceleration;
    arAxisCtrl_gb[AxisNo.OutRobot_Y].PosMode.Jerk := CurrentData.Axes.OutRobot_Y.HalfAuto.Jerk;
    arAxisCtrl_gb[AxisNo.OutRobot_Y].PosMode.Velocity := CurrentData.Axes.OutRobot_Y.HalfAuto.Velocity;		   
    arAxisCtrl_gb[AxisNo.OutRobot_Y].Admin._OpMode.en := ModePosAbs;
ELSIF (AllocateService.AutoMode_BoxMoveReverse.HandShake.Busy 
	  OR AllocateService.AutoMode_EmptyBoxMove.HandShake.Busy 
	  OR AllocateService.AutoMode_RareBoxMove.HandShake.Busy) AND AllowOutRobotMove THEN
	arAxisCtrl_gb[AxisNo.OutRobot_Y].PosMode.Acc := CurrentData.Axes.OutRobot_Y.Auto.Acceleration;
    arAxisCtrl_gb[AxisNo.OutRobot_Y].PosMode.Dec := CurrentData.Axes.OutRobot_Y.Auto.Deceleration;
    arAxisCtrl_gb[AxisNo.OutRobot_Y].PosMode.Jerk := CurrentData.Axes.OutRobot_Y.Auto.Jerk;
    arAxisCtrl_gb[AxisNo.OutRobot_Y].PosMode.Velocity := CurrentData.Axes.OutRobot_Y.Auto.Velocity;		   
    arAxisCtrl_gb[AxisNo.OutRobot_Y].Admin._OpMode.en := ModePosAbs;
ELSE
    arAxisCtrl_gb[AxisNo.OutRobot_Y].Admin.StopDeceleration := 1000;
    arAxisCtrl_gb[AxisNo.OutRobot_Y].Admin._OpMode.en := E_AXIS_MODE.ModeAH;
END_IF

{Endregion}

{region "RoundBelt Axis"}
IF AllocateManualCommand.RoundBelt.Axis.JOG.MoveFWD AND AllowRoundBeltMove THEN
    arAxisCtrl_gb[AxisNo.RoundBelt].VelMode.Acc := CurrentData.Axes.RoundBelt.Manual.JogAcceleration;
    arAxisCtrl_gb[AxisNo.RoundBelt].VelMode.Dec := CurrentData.Axes.RoundBelt.Manual.JogDeceleration;
    arAxisCtrl_gb[AxisNo.RoundBelt].VelMode.Jerk := CurrentData.Axes.RoundBelt.Manual.JogJerk;
    arAxisCtrl_gb[AxisNo.RoundBelt].VelMode.Velocity := CurrentData.Axes.RoundBelt.Manual.JogVelocity;
    arAxisCtrl_gb[AxisNo.RoundBelt].Admin._OpMode.en := E_AXIS_MODE.ModeVel;
ELSIF AllocateManualCommand.RoundBelt.Axis.JOG.MoveBWD AND AllowRoundBeltMove THEN
    arAxisCtrl_gb[AxisNo.RoundBelt].VelMode.Acc := CurrentData.Axes.RoundBelt.Manual.JogAcceleration;
    arAxisCtrl_gb[AxisNo.RoundBelt].VelMode.Dec := CurrentData.Axes.RoundBelt.Manual.JogDeceleration;
    arAxisCtrl_gb[AxisNo.RoundBelt].VelMode.Jerk := CurrentData.Axes.RoundBelt.Manual.JogJerk;
    arAxisCtrl_gb[AxisNo.RoundBelt].VelMode.Velocity := CurrentData.Axes.RoundBelt.Manual.JogVelocity * -1;
    arAxisCtrl_gb[AxisNo.RoundBelt].Admin._OpMode.en := E_AXIS_MODE.ModeVel;
ELSIF AllocateManualCommand.RoundBelt.Axis.PTP.Enable AND AllowRoundBeltMove THEN
    arAxisCtrl_gb[AxisNo.RoundBelt].PosMode.Acc := CurrentData.Axes.RoundBelt.Manual.PtpAcceleration;
    arAxisCtrl_gb[AxisNo.RoundBelt].PosMode.Dec := CurrentData.Axes.RoundBelt.Manual.PtpDeceleration;
    arAxisCtrl_gb[AxisNo.RoundBelt].PosMode.Jerk := CurrentData.Axes.RoundBelt.Manual.PtpJerk;
    arAxisCtrl_gb[AxisNo.RoundBelt].PosMode.Velocity := CurrentData.Axes.RoundBelt.Manual.PtpVelocity;
    arAxisCtrl_gb[AxisNo.RoundBelt].PosMode.Position := CurrentData.Axes.RoundBelt.Manual.PtpPosition;
    arAxisCtrl_gb[AxisNo.RoundBelt].Admin._OpMode.en := ModePosAbs;
ELSIF (AllocateManualCommand.RoundBelt.Axis.Homing.Execute OR  fbAllocateArea.fbAllocateHome.AxisHomingRequest ) AND AllowRoundBeltMove THEN
    arAxisCtrl_gb[AxisNo.RoundBelt].SetupMode.eHomingMode := E_HomingMode._20_Pos_HomeInnerLeft;
    arAxisCtrl_gb[AxisNo.RoundBelt].SetupMode.FastVelo := CurrentData.Axes.RoundBelt.Homing.FastVelo;
    arAxisCtrl_gb[AxisNo.RoundBelt].SetupMode.SlowVelo := CurrentData.Axes.RoundBelt.Homing.SlowVelo;
    arAxisCtrl_gb[AxisNo.RoundBelt].SetupMode.lrOffset := CurrentData.Axes.RoundBelt.Homing.Offset;
    arAxisCtrl_gb[AxisNo.RoundBelt].SetupMode.lrSetPosition := CurrentData.Axes.RoundBelt.Homing.SetAbsolutePosition;
    arAxisCtrl_gb[AxisNo.RoundBelt].SetupMode.stPosBiasParameter.bSetPostionBias := TRUE;
    arAxisCtrl_gb[AxisNo.RoundBelt].Admin._OpMode.en := ModeHoming;
ELSIF TableMove.xBusy AND AllowRoundBeltMove THEN
    arAxisCtrl_gb[AxisNo.RoundBelt].Admin._OpMode.en := ModePosAbs;
ELSIF AllocateService.AllocateCircleMove.HandShake.Busy AND AllowRoundBeltMove THEN
    arAxisCtrl_gb[AxisNo.RoundBelt].PosMode.Acc := CurrentData.Axes.RoundBelt.HalfAuto.Acceleration;
    arAxisCtrl_gb[AxisNo.RoundBelt].PosMode.Dec := CurrentData.Axes.RoundBelt.HalfAuto.Deceleration;
    arAxisCtrl_gb[AxisNo.RoundBelt].PosMode.Jerk := CurrentData.Axes.RoundBelt.HalfAuto.Jerk;
    arAxisCtrl_gb[AxisNo.RoundBelt].PosMode.Velocity := CurrentData.Axes.RoundBelt.HalfAuto.Velocity;
    arAxisCtrl_gb[AxisNo.RoundBelt].Admin._OpMode.en := ModePosAbs;
ELSIF //(AllocateService.AutoMode_AllocateBatchMode.HandShake.Busy OR 
//StorageService.AutoMode_ReloadRoundBeltBoxWithRobot.Status.Busy OR 
//AllocateService.AutoMode_AllocateBatchMode_Reverse.HandShake.Busy) 
THIS^.fbAllocateArea._RoundBeltMoveJob.HandShake.Busy	AND 
	 fbAllocateArea.RoundBeltControl.AxisRoundMoveRequest AND
AllowRoundBeltMove THEN
    arAxisCtrl_gb[AxisNo.RoundBelt].PosMode.Acc := CurrentData.Axes.RoundBelt.HalfAuto.Acceleration;
    arAxisCtrl_gb[AxisNo.RoundBelt].PosMode.Dec := CurrentData.Axes.RoundBelt.HalfAuto.Deceleration;
    arAxisCtrl_gb[AxisNo.RoundBelt].PosMode.Jerk := CurrentData.Axes.RoundBelt.HalfAuto.Jerk;
    arAxisCtrl_gb[AxisNo.RoundBelt].PosMode.Velocity := CurrentData.Axes.RoundBelt.HalfAuto.Velocity;
    arAxisCtrl_gb[AxisNo.RoundBelt].Admin._OpMode.en := ModePosAbs;
//AutoMode Action
ELSIF (AllocateService.AutoMode_AllocateCircleMove.HandShake.Busy OR 
fbAllocateArea.RoundBeltMoveJob_Status.Busy)AND 
	 fbAllocateArea.RoundBeltControl.AxisRoundMoveRequest AND 
AllowRoundBeltMove THEN
    arAxisCtrl_gb[AxisNo.RoundBelt].PosMode.Acc := CurrentData.Axes.RoundBelt.Auto.Acceleration;
    arAxisCtrl_gb[AxisNo.RoundBelt].PosMode.Dec := CurrentData.Axes.RoundBelt.Auto.Deceleration;
    arAxisCtrl_gb[AxisNo.RoundBelt].PosMode.Jerk := CurrentData.Axes.RoundBelt.Auto.Jerk;
    arAxisCtrl_gb[AxisNo.RoundBelt].PosMode.Velocity := CurrentData.Axes.RoundBelt.Auto.Velocity;
    arAxisCtrl_gb[AxisNo.RoundBelt].Admin._OpMode.en := ModePosAbs;
ELSE
    arAxisCtrl_gb[AxisNo.RoundBelt].Admin.StopDeceleration := 1000;
    arAxisCtrl_gb[AxisNo.RoundBelt].Admin._OpMode.en := E_AXIS_MODE.ModeAH;
END_IF

{endregion}

{region "TurnTable Axis"}
IF AllocateManualCommand.TurnTable.Axis.JOG.MoveFWD AND AllowTurnTable THEN
    arAxisCtrl_gb[AxisNo.TurnTable].VelMode.Acc := CurrentData.Axes.TurnTable.Manual.JogAcceleration;
    arAxisCtrl_gb[AxisNo.TurnTable].VelMode.Dec := CurrentData.Axes.TurnTable.Manual.JogDeceleration;
    arAxisCtrl_gb[AxisNo.TurnTable].VelMode.Jerk := CurrentData.Axes.TurnTable.Manual.JogJerk;
    arAxisCtrl_gb[AxisNo.TurnTable].VelMode.Velocity := CurrentData.Axes.TurnTable.Manual.JogVelocity;
    arAxisCtrl_gb[AxisNo.TurnTable].Admin._OpMode.en := E_AXIS_MODE.ModeVel;
ELSIF AllocateManualCommand.TurnTable.Axis.JOG.MoveBWD THEN
    arAxisCtrl_gb[AxisNo.TurnTable].VelMode.Acc := CurrentData.Axes.TurnTable.Manual.JogAcceleration;
    arAxisCtrl_gb[AxisNo.TurnTable].VelMode.Dec := CurrentData.Axes.TurnTable.Manual.JogDeceleration;
    arAxisCtrl_gb[AxisNo.TurnTable].VelMode.Jerk := CurrentData.Axes.TurnTable.Manual.JogJerk;
    arAxisCtrl_gb[AxisNo.TurnTable].VelMode.Velocity := CurrentData.Axes.TurnTable.Manual.JogVelocity * -1;
    arAxisCtrl_gb[AxisNo.TurnTable].Admin._OpMode.en := E_AXIS_MODE.ModeVel;
ELSIF AllocateManualCommand.TurnTable.Axis.PTP.Enable THEN
    arAxisCtrl_gb[AxisNo.TurnTable].PosMode.Acc := CurrentData.Axes.TurnTable.Manual.PtpAcceleration;
    arAxisCtrl_gb[AxisNo.TurnTable].PosMode.Dec := CurrentData.Axes.TurnTable.Manual.PtpDeceleration;
    arAxisCtrl_gb[AxisNo.TurnTable].PosMode.Jerk := CurrentData.Axes.TurnTable.Manual.PtpJerk;
    arAxisCtrl_gb[AxisNo.TurnTable].PosMode.Velocity := CurrentData.Axes.TurnTable.Manual.PtpVelocity;
    arAxisCtrl_gb[AxisNo.TurnTable].PosMode.Position := CurrentData.Axes.TurnTable.Manual.PtpPosition;
    arAxisCtrl_gb[AxisNo.TurnTable].Admin._OpMode.en := ModePosAbs;
ELSIF (AllocateManualCommand.TurnTable.Axis.Homing.Execute OR  fbAllocateArea.fbAllocateHome.AxisHomingRequest) AND  AllowTurnTable THEN
    arAxisCtrl_gb[AxisNo.TurnTable].SetupMode.eHomingMode := E_HomingMode._22_Neg_HomeInnerRight;
    arAxisCtrl_gb[AxisNo.TurnTable].SetupMode.FastVelo := CurrentData.Axes.TurnTable.Homing.FastVelo;
    arAxisCtrl_gb[AxisNo.TurnTable].SetupMode.SlowVelo := CurrentData.Axes.TurnTable.Homing.SlowVelo;
    arAxisCtrl_gb[AxisNo.TurnTable].SetupMode.lrOffset := CurrentData.Axes.TurnTable.Homing.Offset;
    arAxisCtrl_gb[AxisNo.TurnTable].SetupMode.lrSetPosition := CurrentData.Axes.TurnTable.Homing.SetAbsolutePosition;
    arAxisCtrl_gb[AxisNo.TurnTable].SetupMode.stPosBiasParameter.bSetPostionBias := TRUE;
    arAxisCtrl_gb[AxisNo.TurnTable].Admin._OpMode.en := ModeHoming;
ELSIF TableMove.xBusy AND AllowTurnTable THEN
    arAxisCtrl_gb[AxisNo.TurnTable].Admin._OpMode.en := ModePosAbs;
ELSIF (AllocateService.TurnTableMove.HandShake.Busy ) AND fbAllocateArea.TurnTableControl.bTurnTableMoveRequest AND AllowTurnTable THEN
    arAxisCtrl_gb[AxisNo.TurnTable].PosMode.Acc := CurrentData.Axes.TurnTable.HalfAuto.Acceleration;
    arAxisCtrl_gb[AxisNo.TurnTable].PosMode.Dec := CurrentData.Axes.TurnTable.HalfAuto.Deceleration;
    arAxisCtrl_gb[AxisNo.TurnTable].PosMode.Jerk := CurrentData.Axes.TurnTable.HalfAuto.Jerk;
    arAxisCtrl_gb[AxisNo.TurnTable].PosMode.Velocity := CurrentData.Axes.TurnTable.HalfAuto.Velocity;
    arAxisCtrl_gb[AxisNo.TurnTable].Admin._OpMode.en := ModePosAbs;
ELSIF AllocateService.AutoMode_TurnTableMove.HandShake.Busy AND fbAllocateArea.TurnTableControl.bTurnTableMoveRequest AND AllowTurnTable THEN
    arAxisCtrl_gb[AxisNo.TurnTable].PosMode.Acc := CurrentData.Axes.TurnTable.Auto.Acceleration;
    arAxisCtrl_gb[AxisNo.TurnTable].PosMode.Dec := CurrentData.Axes.TurnTable.Auto.Deceleration;
    arAxisCtrl_gb[AxisNo.TurnTable].PosMode.Jerk := CurrentData.Axes.TurnTable.Auto.Jerk;
    arAxisCtrl_gb[AxisNo.TurnTable].PosMode.Velocity := CurrentData.Axes.TurnTable.Auto.Velocity;
    arAxisCtrl_gb[AxisNo.TurnTable].Admin._OpMode.en := ModePosAbs;
ELSE
    arAxisCtrl_gb[AxisNo.TurnTable].Admin.StopDeceleration := 1000;
    arAxisCtrl_gb[AxisNo.TurnTable].Admin._OpMode.en := E_AXIS_MODE.ModeAH;
END_IF

{endregion}


IF NOT (fbStorageArea.RackState = E_RackState.FeedBox) AND 
	NOT (fbStorageArea.RackState = E_RackState.TransitingFeedBox) OR 
	fbStorageArea.fbStorageHoming.xBusy THEN
			
		IF StorageManualCommand.RackMotor.Axis.JOG.MoveFWD AND AllowRackMotor THEN
			arAxisCtrl_gb[AxisNo.RackMotor].VelMode.Acc := CurrentData.Axes.RackMotor.Manual.JogAcceleration;
			arAxisCtrl_gb[AxisNo.RackMotor].VelMode.Dec := CurrentData.Axes.RackMotor.Manual.JogDeceleration;
			arAxisCtrl_gb[AxisNo.RackMotor].VelMode.Jerk := CurrentData.Axes.RackMotor.Manual.JogJerk;
			arAxisCtrl_gb[AxisNo.RackMotor].VelMode.Velocity := CurrentData.Axes.RackMotor.Manual.JogVelocity;
			arAxisCtrl_gb[AxisNo.RackMotor].Admin._OpMode.en := E_AXIS_MODE.ModeVel;
		ELSIF StorageManualCommand.RackMotor.Axis.JOG.MoveBWD AND AllowRackMotor THEN
			arAxisCtrl_gb[AxisNo.RackMotor].VelMode.Acc := CurrentData.Axes.RackMotor.Manual.JogAcceleration;
			arAxisCtrl_gb[AxisNo.RackMotor].VelMode.Dec := CurrentData.Axes.RackMotor.Manual.JogDeceleration;
			arAxisCtrl_gb[AxisNo.RackMotor].VelMode.Jerk := CurrentData.Axes.RackMotor.Manual.JogJerk;
			arAxisCtrl_gb[AxisNo.RackMotor].VelMode.Velocity := CurrentData.Axes.RackMotor.Manual.JogVelocity * -1;
			arAxisCtrl_gb[AxisNo.RackMotor].Admin._OpMode.en := E_AXIS_MODE.ModeVel;
		ELSIF StorageManualCommand.RackMotor.Axis.PTP.Enable AND AllowRackMotor THEN
			arAxisCtrl_gb[AxisNo.RackMotor].PosMode.Acc := CurrentData.Axes.RackMotor.Manual.PtpAcceleration;
			arAxisCtrl_gb[AxisNo.RackMotor].PosMode.Dec := CurrentData.Axes.RackMotor.Manual.PtpDeceleration;
			arAxisCtrl_gb[AxisNo.RackMotor].PosMode.Jerk := CurrentData.Axes.RackMotor.Manual.PtpJerk;
			arAxisCtrl_gb[AxisNo.RackMotor].PosMode.Velocity := CurrentData.Axes.RackMotor.Manual.PtpVelocity;
			arAxisCtrl_gb[AxisNo.RackMotor].PosMode.Position := CurrentData.Axes.RackMotor.Manual.PtpPosition;
			arAxisCtrl_gb[AxisNo.RackMotor].Admin._OpMode.en := ModePosAbs;
		ELSIF (StorageManualCommand.RackMotor.Axis.Homing.Execute OR fbStorageArea.fbStorageHoming.RackMotorHomeRequest) AND AllowRackMotor THEN
			arAxisCtrl_gb[AxisNo.RackMotor].SetupMode.eHomingMode := E_HomingMode._17_Neg_LimitOutterRight;
			arAxisCtrl_gb[AxisNo.RackMotor].SetupMode.FastVelo := CurrentData.Axes.RackMotor.Homing.FastVelo;
			arAxisCtrl_gb[AxisNo.RackMotor].SetupMode.SlowVelo := CurrentData.Axes.RackMotor.Homing.SlowVelo;
			arAxisCtrl_gb[AxisNo.RackMotor].SetupMode.lrOffset := CurrentData.Axes.RackMotor.Homing.Offset;
			arAxisCtrl_gb[AxisNo.RackMotor].SetupMode.lrSetPosition := CurrentData.Axes.RackMotor.Homing.SetAbsolutePosition;
			arAxisCtrl_gb[AxisNo.RackMotor].SetupMode.stPosBiasParameter.bSetPostionBias := TRUE;
			arAxisCtrl_gb[AxisNo.RackMotor].Admin._OpMode.en := ModeHoming;
		ELSIF (TableMove.xBusy OR StorageService.AutoMode_AddBoxes.Status.Busy) AND AllowRackMotor THEN
			arAxisCtrl_gb[AxisNo.RackMotor].Admin._OpMode.en := ModePosAbs;
		ELSE
			arAxisCtrl_gb[AxisNo.RackMotor].Admin.StopDeceleration := 1000;
			arAxisCtrl_gb[AxisNo.RackMotor].Admin._OpMode.en := E_AXIS_MODE.ModeAH;
		END_IF
ELSIF fbStorageArea.fbBoxSupplyCtrl.Busy AND 
			fbStorageArea.fbBoxSupplyCtrl.AxisRackMotorBTNHomeRequest AND 
			AllowRackMotor THEN
		arAxisCtrl_gb[AxisNo.RackMotor].PosMode.Acc := CurrentData.Axes.RackMotor.HalfAuto.Acceleration;
		arAxisCtrl_gb[AxisNo.RackMotor].PosMode.Dec := CurrentData.Axes.RackMotor.HalfAuto.Deceleration;
		arAxisCtrl_gb[AxisNo.RackMotor].PosMode.Jerk := CurrentData.Axes.RackMotor.HalfAuto.Jerk;
		arAxisCtrl_gb[AxisNo.RackMotor].PosMode.Velocity := CurrentData.Axes.RackMotor.HalfAuto.Velocity;
		arAxisCtrl_gb[AxisNo.RackMotor].Admin._OpMode.en := ModePosAbs;	  
ELSE
		arAxisCtrl_gb[AxisNo.RackMotor].Admin.StopDeceleration := 1000;
		arAxisCtrl_gb[AxisNo.RackMotor].Admin._OpMode.en := E_AXIS_MODE.ModeAH;	 
END_IF
END_METHOD

METHOD M_Clearing
VAR
	CylinderIndex : UDINT;
	MotorIndex : INT;
	ServoIndex : INT;
END_VAR
VAR_INST
	AllCylinderNoError : BOOL := TRUE;
	AllMotorNoError : BOOL := TRUE;
	AllServoNoError : BOOL := TRUE;
END_VAR
// Disable all cylinder 
FOR CylinderIndex := 1 TO udiMax_CylinderNum DO
    Cylinder.arCylinder[CylinderIndex].xEnable := FALSE;
END_FOR

// Disable all motor
FOR MotorIndex := 1 TO 26 DO
    Motor.arMotor[MotorIndex].xEnable := FALSE;
END_FOR

// Check cylinder no error
FOR CylinderIndex := 1 TO udiMax_CylinderNum DO
    IF Cylinder.arCylinder[CylinderIndex].xError THEN
        AllCylinderNoError := FALSE;
        EXIT;
    END_IF
END_FOR

// Check motor no error
FOR MotorIndex := 1 TO 26 DO
    IF Motor.arMotor[MotorIndex].xError THEN
        AllMotorNoError := FALSE;
        EXIT;
    END_IF
END_FOR

FOR ServoIndex := 1 TO 7 DO
	IF arAxisCtrl_gb[ServoIndex].Admin.Axis.Status.Error THEN
		arAxisCtrl_gb[ServoIndex].Admin.ClearError := TRUE;
	END_IF
END_FOR
AllServoNoError := TRUE;
FOR ServoIndex := 1 TO 7 DO
    IF arAxisCtrl_gb[ServoIndex].Admin.Axis.Status.Error THEN
        AllServoNoError := FALSE;
        EXIT;
    END_IF
END_FOR
CASE eModeCurrent OF
    E_UnitMode.Manual:
        GVL_Machine.PackTags[UnitNo.Allocate].Command.UnitMode := E_UnitMode.Manual;
        GVL_Machine.PackTags[UnitNo.Allocate].Command.CntrlCmd := ePMLCommand_Clear;
        GVL_Machine.PackTags[UnitNo.Storage].Command.UnitMode := E_UnitMode.Manual;
        GVL_Machine.PackTags[UnitNo.Storage].Command.CntrlCmd := ePMLCommand_Clear;
        GVL_Machine.PackTags[UnitNo.Shipping].Command.UnitMode := E_UnitMode.Manual;
        GVL_Machine.PackTags[UnitNo.Shipping].Command.CntrlCmd := ePMLCommand_Clear;

        IF GVL_Machine.PackTags[UnitNo.Allocate].Status.StateCurrent = ePMLState_Stopped AND
            GVL_Machine.PackTags[UnitNo.Storage].Status.StateCurrent = ePMLState_Stopped AND
            GVL_Machine.PackTags[UnitNo.Shipping].Status.StateCurrent = ePMLState_Stopped THEN
            IF AllCylinderNoError AND AllMotorNoError AND AllServoNoError THEN
                M_StateComplete();
            END_IF
        END_IF

    E_UnitMode.Auto: ;
        GVL_Machine.PackTags[UnitNo.Allocate].Command.UnitMode := E_UnitMode.Auto;
        GVL_Machine.PackTags[UnitNo.Allocate].Command.CntrlCmd := ePMLCommand_Clear;
        GVL_Machine.PackTags[UnitNo.Storage].Command.UnitMode := E_UnitMode.Auto;
        GVL_Machine.PackTags[UnitNo.Storage].Command.CntrlCmd := ePMLCommand_Clear;
        GVL_Machine.PackTags[UnitNo.Shipping].Command.UnitMode := E_UnitMode.Auto;
        GVL_Machine.PackTags[UnitNo.Shipping].Command.CntrlCmd := ePMLCommand_Clear;

        IF GVL_Machine.PackTags[UnitNo.Allocate].Status.StateCurrent = ePMLState_Stopped AND
            GVL_Machine.PackTags[UnitNo.Storage].Status.StateCurrent = ePMLState_Stopped AND
            GVL_Machine.PackTags[UnitNo.Shipping].Status.StateCurrent = ePMLState_Stopped THEN
            IF AllCylinderNoError AND AllMotorNoError AND AllServoNoError THEN
                M_StateComplete();
            END_IF
        END_IF
END_CASE
END_METHOD

METHOD PRIVATE M_ClearOutput : BOOL
VAR_INPUT
END_VAR
VAR
	SpaceOutput : ST_OutputTable;
END_VAR
OUTPUT := SpaceOutput;
M_ClearOutput := true;
END_METHOD

METHOD M_Complete
M_StateComplete();
END_METHOD

METHOD M_Completing
M_StateComplete();
END_METHOD

METHOD M_Execute
VAR
	CylinderIndex : UDINT;
	MotorIndex    : INT;
END_VAR
//M_StateComplete();
// 啟用汽缸和馬達（從 M_Resetting 移至此處，避免 Resetting ↔ Aborting 循環導致汽缸來回往復）
FOR CylinderIndex := 1 TO udiMax_CylinderNum DO
    Cylinder.arCylinder[CylinderIndex].xEnable := TRUE;
END_FOR
FOR MotorIndex := 1 TO 26 DO
    Motor.arMotor[MotorIndex].xEnable := TRUE;
END_FOR

CASE eModeCurrent OF
    E_UnitMode.Manual:
			M_Manual_Cylinder();
			M_Manual_Axes();
			M_Manual_Motor();
			M_HalfAuto_TableMove();
			IF NOT fbMachineHoming.xBusy THEN
				M_ManualAllocateHoming();
				M_ManualStorageHoming();
				M_ManualShippingHoming();
			END_IF
			M_ManualMachineHome();
			
    E_UnitMode.Auto:
			M_Auto_Axes();
  
END_CASE
//fbAllocateArea.A00_Service();
M_StroageRobotSafeCheck();
IF ErrorTableInitDone THEN
	M_General_AlarmRegister();
END_IF
END_METHOD

METHOD M_General_AlarmRegister : BOOL
VAR_INPUT
END_VAR
VAR
END_VAR
VAR_INST
	bTest 		  : ARRAY[1..200] OF BOOL;
	bByPassModBusRTU	: ARRAY[1..4] OF BOOL;
	bFanucStoTrig		: ARRAY[1..17] OF BOOL;	// 大手臂 detail alarm trigger 160-176 (RegisterAlarm.Trigger 是 VAR_IN_OUT 不能塞表達式)
	bFanucShpTrig		: ARRAY[1..17] OF BOOL;	// 小手臂 detail alarm trigger 180-196
END_VAR
/////  Category ==> 0 :machine Area ,1: StorageArea ,2: AllocateArea ,3: ShippingArea 

// E-Stop
RegisterAlarm(Trigger := Allocate_Estop, 								ID := 001,value := E_Severity.Level7, Message := GVL_ErrorCode.GC_MSG_0176, Category := 2);
RegisterAlarm(Trigger := Storage_EStop, 								ID := 002,value := E_Severity.Level7, Message := GVL_ErrorCode.GC_MSG_0177, Category := 1);
RegisterAlarm(Trigger := FanucRobot.List.StorageRobot.E_Stop_Output,	ID := 003,value := E_Severity.Level7,Message := GVL_ErrorCode.GC_MSG_0178,Category := 1);
RegisterAlarm(Trigger := FanucRobot.List.ShippingRobot.E_Stop_Output,	ID := 004,value := E_Severity.Level7,Message := GVL_ErrorCode.GC_MSG_0179,Category := 1);

//AirPressure
bStorage_AirPressure := NOT( BIT_TO_BOOL( INPUT.bStorage_AirPressure_Ready) ) OR  bTest2;
RegisterAlarm(Trigger := bStorage_AirPressure,							ID := 005,value := E_Severity.Level7,Message := GVL_ErrorCode.GC_MSG_0180,Category := 1);


//Homing Service
RegisterAlarm(Trigger := fbMachineHoming.xError,				ID := GVL_ErrorCode.GC_ALARM_MACHINE_HOMING,value := E_Severity.Level4,Message := fbMachineHoming.ErrorMsg,Category := 0);
RegisterAlarm(Trigger := fbStorageArea.fbStorageHoming.xError,	ID := GVL_ErrorCode.GC_ALARM_STORAGE_HOMING,value := E_Severity.Level4,Message := fbStorageArea.fbStorageHoming.ErrorMsg,Category := 1);
RegisterAlarm(Trigger := fballocateArea.fballocateHome.xError,	ID := GVL_ErrorCode.GC_ALARM_ALLOCATE_HOMING,value := E_Severity.Level4,Message := fballocateArea.fballocateHome.ErrorMsg,Category := 2);
RegisterAlarm(Trigger := fbShippingArea.fbShippingHoming.xError,ID := GVL_ErrorCode.GC_ALARM_SHIPPING_HOMING,value := E_Severity.Level4,Message := fbShippingArea.fbShippingHoming.ErrorMsg,Category := 3);
//Machine Area Service
RegisterAlarm(Trigger := TableMove.xError , 					ID := GVL_ErrorCode.GC_ALARM_TABLE_MOVE,value := E_Severity.Level4,Message := TableMove.ErrorMsg,Category := 2);
RegisterAlarm(Trigger := fbMachineModeSwitch.Error , 			ID := GVL_ErrorCode.GC_ALARM_MACHINEMODE_SWITCH,value := E_Severity.Level4,Message := fbMachineModeSwitch.Status,Category := 2);


